  4071 = 'RESET REMAINING\nDOSING VOLUME (ml)' | German: 'RESET RESTDOSIERVOLUMEN (ml)' | France: 'RESET VOLUME DE DOSAGE RESTANT (ml)' | English: 'RESET REMAINING\nDOSING VOLUME (ml)'
  7600 = 'RIGHT\nBOTTOM' | German: 'RECHTS UNTEN' | France: 'DROITE EN BAS' | English: 'RIGHT\nBOTTOM'
  3413 = 'RIGHT\nTOP' | German: 'RECHTS OBEN' | France: 'DROITE EN HAUT' | English: 'RIGHT\nTOP'
  6630 = 'RIGHT BOTTOM TEMP (°C) ' | German: 'TEMPERATUR UNTEN RECHTS' | France: 'TEMPÉRATURE EN BAS À DROITE (?C)' | English: 'RIGHT BOTTOM TEMP (°C) '
  7664 = 'RIGHT TOP TEMP (°C) ' | German: 'TEMPERATUR OBEN RECHTS' | France: 'TEMPÉRATURE EN HAUT À DROITE (?C)' | English: 'RIGHT TOP TEMP (°C) '
  3245 = 'ROTARY BARREL' | German: 'TROMMEL' | France: 'BARILLET ROTATIF' | English: 'ROTARY BARREL'
  4283 = 'ROTARY BARREL - ROBOT' | German: 'TROMMEL - ROTATIONSROBOTER' | France: 'BARILLET ROTATIF - ROBOT DE ROTATION' | English: 'ROTARY BARREL - ROBOT'
  7424 = 'ROTARY BARREL - STATION' | German: 'TROMMEL - WANNE' | France: 'BARILLET ROTATIF - CUVE' | English: 'ROTARY BARREL - STATION'
  2002 = 'ROTATING BARREL' | German: 'TROMMEL' | France: 'BARILLET ROTATIF' | English: 'ROTATING BARREL'
  374 = 'ROW LOADING INC AV-3' | English: 'ROW LOADING INC AV-3'
  6590 = 'ROW MAIN INC AV-2' | English: 'ROW MAIN INC AV-2'
  254 = 'RUN' | German: 'RUN' | France: 'MARCHE' | English: 'RUN'
  5034 = 'SATURDAY' | German: 'SAMSTAG' | France: 'SAMEDI' | English: 'SATURDAY'
  53 = 'SAVE' | German: 'SPEICHERN' | France: 'ENREGISTRER' | English: 'SAVE'
  667 = 'Scan Complete' | German: 'Scan abgeschlossen' | France: 'Scan terminé' | English: 'Scan Complete'
  447 = 'Scan Start' | German: 'Start des Scans' | France: 'Démarrage du scan' | English: 'Scan Start'
  4578 = 'SENSOR A MISSHOOK\nALARM DEACTIVATED' | German: 'SENSOR A FEHLHAKEN\nALARM DEAKTIVIERT' | France: 'DÉTECTEUR A MAL ACCROCHÉ\nALARME DÉSACTIVÉE' | English: 'SENSOR A MISSHOOK\nALARM DEACTIVATED'
  3015 = 'SENSOR B MISSHOOK\nALARM DEACTIVATED' | German: 'SENSOR B FEHLHAKEN\nALARM DEAKTIVIERT' | France: 'DÉTECTEUR B MAL ACCROCHÉ\nALARME DÉSACTIVÉE' | English: 'SENSOR B MISSHOOK\nALARM DEACTIVATED'
  4042 = 'SEQUENCE RECIPE CONFIGURATION (SSER)' | German: 'KONFIGURATION DER SEQUENZREZEPTE (SSER)' | France: 'CONFIGURATION DE LA RECETTE DE SÉQUENCE (SSER)' | English: 'SEQUENCE RECIPE CONFIGURATION (SSER)'
  1305 = 'SEQUENCE RECIPE INFO (SSER)' | German: 'SEQUENZ REZEPTINFO (SSER)' | France: 'INFORMATION SUR LA RECETTE DE LA SÉQUENCE (SSER)' | English: 'SEQUENCE RECIPE INFO (SSER)'
  3694 = 'SET TIME' | German: 'SOLLZEIT' | France: 'TEMPS DE CONSIGNE' | English: 'SET TIME'
  1659 = 'SET VALUE' | German: 'WERT EINSTELLEN' | France: 'DEFINITION DES VALEURS' | English: 'SET VALUE'
  197 = 'SETTING' | German: 'EINSTELLUNG' | France: 'PARAMÈTRES' | English: 'SETTING'
  669 = 'SLOWPULL' | German: 'LIFT OUT' | France: 'SORTIE LENTE' | English: 'SLOWPULL'
  2167 = 'SLOWPULL\nDOWN' | German: 'LIFT OUT\nNACH UNTEN' | France: 'SORTIE LENTE\nNEN BAS' | English: 'SLOWPULL\nDOWN'
  3255 = 'SLOWPULL\nUP' | German: 'LIFT OUT\nNACH ' | France: 'SORTIE LENTE\nHAUT' | English: 'SLOWPULL\nUP'
  4405 = 'SLOWPULL DOWN STN 8' | German: 'LANGSAMES ZIEHEN NACH UNTEN WANNE 8' | France: 'RALENTISSEMENT DE LA DESCENTE AU POSTE 8' | English: 'SLOWPULL DOWN STN 8'
  3314 = 'SLOWPULL JOG VELO (mm/s)' | English: 'SLOWPULL JOG VELO (mm/s)'
  4447 = 'SLOWPULL POSITION' | English: 'SLOWPULL POSITION'
  2433 = 'SLOWPULL VELOCITY (mm/s)' | English: 'SLOWPULL VELOCITY (mm/s)'
  4890 = 'SPEED PATTERN NO' | German: 'GESCHWINDIGKEIT MUSTERNUMMER' | France: 'VITESSE ENTRE POSITION' | English: 'SPEED PATTERN NO'
  4281 = 'SPEED PROFILE NO.' | German: 'GESCHWINDIGKEIT PROFILNUMMER' | France: 'NUMERO DU TYPE DE VITESSE' | English: 'SPEED PROFILE NO.'
  4424 = 'SSER' | German: 'SSER' | France: 'SSER' | English: 'SSER'
  3904 = 'SSER NAME' | German: 'SSER NAME' | France: 'SSER NAME' | English: 'SSER NAME'
  4062 = 'SSER NO.' | German: 'SSER NO.' | France: 'SSER NO.' | English: 'SSER NO.'
  646 = 'SSUR' | German: 'SSUR' | France: 'SSUR' | English: 'SSUR'
  1459 = 'SSUR NAME' | German: 'SSUR NAME' | France: 'SSUR NAME' | English: 'SSUR NAME'
  1820 = 'SSUR NO.' | German: 'SSUR NO.' | France: 'SSUR NO.' | English: 'SSUR NO.'
  224 = 'START' | German: 'START' | France: 'DEMARRER' | English: 'START'
  183 = 'STATION' | German: 'WANNE' | France: 'CUVE' | English: 'STATION'
  370 = 'STATION 01' | German: 'WANNE 01' | France: 'CUVE 01' | English: 'STATION 01'
  742 = 'STATION 02' | German: 'WANNE 02' | France: 'CUVE 02' | English: 'STATION 02'
  859 = 'STATION 03' | German: 'WANNE 03' | France: 'CUVE 03' | English: 'STATION 03'
  200 = 'STATION 04' | German: 'WANNE 04' | France: 'CUVE 04' | English: 'STATION 04'
  72 = 'STATION 05' | German: 'WANNE 05' | France: 'CUVE 05' | English: 'STATION 05'
  509 = 'STATION 06' | German: 'WANNE 06' | France: 'CUVE 06' | English: 'STATION 06'
  120 = 'STATION 07' | German: 'WANNE 07' | France: 'CUVE 07' | English: 'STATION 07'
  712 = 'STATION 08' | German: 'WANNE 08' | France: 'CUVE 08' | English: 'STATION 08'
  1915 = 'STATION 09' | German: 'WANNE 09' | France: 'CUVE 09' | English: 'STATION 09'
  4945 = 'STATION 5 INCOMING WATER' | German: 'WANNE 05 EINGANG VERSORGUNG FÜR WASSER' | France: 'CUVE 05 ALIMENTATION EN EAU ' | English: 'STATION 5 INCOMING WATER'
  3 = 'STATION INFO' | German: 'INFO WANNE' | France: 'INFORMATIONS SUR LA CUVE' | English: 'STATION INFO'
  4252 = 'STATION ROTATION\nBASKET'
  2249 = 'STATION VIEW' | German: 'STATION ANSICHT' | France: 'VUE DE LA STATION' | English: 'STATION VIEW'
  1600 = 'STEP' | German: 'SCHRITTE' | France: 'ETAPE' | English: 'STEP'
  1308 = 'STEP 01' | German: 'SCHRITTE 01' | France: 'ETAPE 01' | English: 'STEP 01'
  541 = 'STEP 02' | German: 'SCHRITTE 02' | France: 'ETAPE 02' | English: 'STEP 02'
  535 = 'STEP 03' | German: 'SCHRITTE 03' | France: 'ETAPE 03' | English: 'STEP 03'
  398 = 'STEP 04' | German: 'SCHRITTE 04' | France: 'ETAPE 04' | English: 'STEP 04'
  1687 = 'STEP 05' | German: 'SCHRITTE 05' | France: 'ETAPE 05' | English: 'STEP 05'
  1286 = 'STEP 06' | German: 'SCHRITTE 06' | France: 'ETAPE 06' | English: 'STEP 06'
  2151 = 'STEP 07' | German: 'SCHRITTE 07' | France: 'ETAPE 07' | English: 'STEP 07'
  1635 = 'STEP 08' | German: 'SCHRITTE 08' | France: 'ETAPE 08' | English: 'STEP 08'
  2165 = 'STEP 09' | German: 'SCHRITTE 09' | France: 'ETAPE 09' | English: 'STEP 09'
  510 = 'STEP 10' | German: 'SCHRITTE 10' | France: 'ETAPE 10' | English: 'STEP 10'
  2122 = 'STEP 11' | German: 'SCHRITTE 11' | France: 'ETAPE 11' | English: 'STEP 11'
  1601 = 'STEP 12' | German: 'SCHRITTE 12' | France: 'ETAPE 12' | English: 'STEP 12'
  1643 = 'STEP 13' | German: 'SCHRITTE 13' | France: 'ETAPE 13' | English: 'STEP 13'
  179 = 'STEP 14' | German: 'SCHRITTE 14' | France: 'ETAPE 14' | English: 'STEP 14'
  2188 = 'STEP 15' | German: 'SCHRITTE 15' | France: 'ETAPE 15' | English: 'STEP 15'
  201 = 'STEP 16' | German: 'SCHRITTE 16' | France: 'ETAPE 16' | English: 'STEP 16'
  1624 = 'STEP 17' | German: 'SCHRITTE 17' | France: 'ETAPE 17' | English: 'STEP 17'
  2332 = 'STEP 18' | German: 'SCHRITTE 18' | France: 'ETAPE 18' | English: 'STEP 18'
  960 = 'STEP 19' | German: 'SCHRITTE 19' | France: 'ETAPE 19' | English: 'STEP 19'
  2078 = 'STEP 20' | German: 'SCHRITTE 20' | France: 'ETAPE 20' | English: 'STEP 20'
  294 = 'STN 01' | German: 'WANNE 01' | France: 'CUVE 01' | English: 'STN 01'
  512 = 'STN 01\nDOWN' | German: 'WANNE 01\nNACH UNTEN' | France: 'CUVE 01\nEN BAS' | English: 'STN 01\nDOWN'
  3517 = 'STN 01\nHOOK' | German: 'WANNE 01\nHAKEN' | France: 'CUVE 01\nACCROCHAGE' | English: 'STN 01\nHOOK'
  2972 = 'STN 01\nUNHOOK' | German: 'WANNE 01\nAUSHANGEN' | France: 'CUVE 01\nDECROCHAGE' | English: 'STN 01\nUNHOOK'
  1354 = 'STN 01 BOTTOM\nSUCTION VALVE AV1-3' | German: 'WANNE 01 DRUCKTASTER\nSAUGLUFTVENTIL 1-3' | France: "CUVE 01 BOUTON-POUSSOIR\nSOUPAPE D'AIR\nD'ASPIRATION 1-3" | English: 'STN 01 BOTTOM\nSUCTION VALVE AV1-3'
  3860 = 'STN 01 BOTTOM\nSUCTION VALVE AV2-3' | German: 'WANNE 01 DRUCKTASTER SAUGLUFTVENTIL 2-3' | France: "CUVE 01 BOUTON-POUSSOIR SOUPAPE D'AIR D'ASPIRATION 2-3" | English: 'STN 01 BOTTOM\nSUCTION VALVE AV2-3'
  8043 = 'STN 01 DIW INC\nSUPPLY VALVE AV1-1' | German: 'WANNE 01 DIW INC\nZUFUHRVENTIL AV1-1' | France: "CUVE 01 DIW INC\nSOUPAPE D'ALIMENTATION\nAV1-1" | English: 'STN 01 DIW INC\nSUPPLY VALVE AV1-1'
  2314 = 'STN 01 DIW INC\nSUPPLY VALVE AV2-1' | German: 'WANNE 01 DIW INC ZUFUHRVENTIL AV2-1' | France: "CUVE 01 DIW INC SOUPAPE D'ALIMENTATION AV2-1" | English: 'STN 01 DIW INC\nSUPPLY VALVE AV2-1'
  474 = 'STN 01 DRAIN' | German: 'WANNE 01 ENTLEERUNG' | France: 'CUVE 01 VIDANGE' | English: 'STN 01 DRAIN'
  1834 = 'STN 01 DRAIN\nVALVE AV1-4' | German: 'WANNE 01 ENTLEERUNG\nSAUGLUFTVENTIL 1-4' | France: "CUVE 01 VIDANGE VANNE\nD'AIR D'ASPIRATION\n1-4" | English: 'STN 01 DRAIN\nVALVE AV1-4'
  1064 = 'STN 01 DRAIN \nVALVE AV1-4' | German: 'WANNE 01 ENTLEERUNG SAUGLUFTVENTIL 1-4' | France: "CUVE 01 VIDANGE VANNE D'AIR D'ASPIRATION 1-4" | English: 'STN 01 DRAIN \nVALVE AV1-4'
  3372 = 'STN 01 DRAIN \nVALVE AV2-4' | German: 'WANNE 01 ENTLEERUNG SAUGLUFTVENTIL 2-4' | France: "CUVE 01 VIDANGE VANNE D'AIR D'ASPIRATION 2-4" | English: 'STN 01 DRAIN \nVALVE AV2-4'
  2307 = 'STN 01 DRAIN  VALVE AV1-4' | German: 'WANNE 01 ENTLEERUNG SAUGLUFTVENTIL 1-4' | France: "CUVE 01 VIDANGE VANNE D'AIR D'ASPIRATION 1-4" | English: 'STN 01 DRAIN  VALVE AV1-4'
  6607 = 'STN 01 DRAIN VALVE AV1-3' | German: 'WANNE 01 ENTLEERUNG\nSAUGLUFTVENTIL 1-3' | France: "CUVE 01 VIDANGE VANNE\nD'AIR D'ASPIRATION 1-3" | English: 'STN 01 DRAIN VALVE AV1-3'
  4935 = 'STN 01 DRAIN VALVE AV1-4' | German: 'WANNE 01 ENTLEERUNG\nSAUGLUFTVENTIL 1-4' | France: "CUVE 01 VIDANGE VANNE\nD'AIR D'ASPIRATION 1-4" | English: 'STN 01 DRAIN VALVE AV1-4'
  4000 = 'STN 01 OVERFLOW\nSUCTION VALVE AV1-2' | German: 'WANNE 01 ÜBERFLUß\nAASAUGUNG VENTIL AV1-2' | France: 'CUVE 01 TROP-PLEIN\nASPIRATION VANNE AV1-2' | English: 'STN 01 OVERFLOW\nSUCTION VALVE AV1-2'
  4585 = 'STN 01 OVERFLOW\nSUCTION VALVE AV2-2' | German: 'WANNE 01 ÜBERFLUß AASAUGUNG VENTIL AV2-3' | France: 'CUVE 01 TROP-PLEIN ASPIRATION VANNE AV2-3' | English: 'STN 01 OVERFLOW\nSUCTION VALVE AV2-2'
  1115 = 'STN 01 PROCESS TANK MIN LEVEL' | German: 'Wanne 01 Niveausensor Prozess - Niveau Minimum' | France: 'CUVE 1 NIVEAU BAS' | English: 'STN 01 PROCESS TANK MIN LEVEL'
  1803 = 'STN 01 READY TEMPERATURE' | German: 'Wanne 01 Bereitschaftstemperatur' | France: 'Cuve 01 Température De Fonctionnement' | English: 'STN 01 READY TEMPERATURE'
  1651 = 'STN 02' | German: 'WANNE 02' | France: 'CUVE 02' | English: 'STN 02'
  2317 = 'STN 02\nDOWN' | German: 'WANNE 02\nNACH UNTEN' | France: 'CUVE 02\nEN BAS' | English: 'STN 02\nDOWN'
  2785 = 'STN 02\nHOOK' | German: 'WANNE 02\nHAKEN' | France: 'CUVE 02\nACCROCHAGE' | English: 'STN 02\nHOOK'
  3442 = 'STN 02\nUNHOOK' | German: 'WANNE 02\nAUSHANGEN' | France: 'CUVE 02\nDECROCHAGE' | English: 'STN 02\nUNHOOK'
  6777 = 'STN 02 BOTTOM\nSUCTION VALVE AV2-3' | German: 'WANNE 02 DRUCKTASTER\nSAUGLUFTVENTIL 2-3' | France: "CUVE 02 BOUTON-POUSSOIR\nSOUPAPE D'AIR\nD'ASPIRATION 2-3" | English: 'STN 02 BOTTOM\nSUCTION VALVE AV2-3'
  3146 = 'STN 02 BOTTOM\nSUCTION VALVE AV2-4' | German: 'WANNE 02 DRUCKTASTER\nSAUGLUFTVENTIL 2-4' | France: "CUVE 02 BOUTON-POUSSOIR\nSOUPAPE D'AIR D'ASPIRATION 2-4" | English: 'STN 02 BOTTOM\nSUCTION VALVE AV2-4'
  731 = 'STN 02 DIW INC\nSUPPLY VALVE AV2-1' | German: 'WANNE 02 DIW INC\nZUFUHRVENTIL AV2-1' | France: "CUVE 02 DIW INC\nSOUPAPE D'ALIMENTATION\nAV2-1" | English: 'STN 02 DIW INC\nSUPPLY VALVE AV2-1'
  4357 = 'STN 02 DRAIN\nVALVE AV2-4' | German: 'WANNE 02 ENTLEERUNG\nSAUGLUFTVENTIL 2-4' | France: "CUVE 02 VIDANGE VANNE\nD'AIR D'ASPIRATION 2-4" | English: 'STN 02 DRAIN\nVALVE AV2-4'
  341 = 'STN 02 DRAIN \nVALVE AV2-4' | German: 'WANNE 02 ENTLEERUNG\nSAUGLUFTVENTIL 2-4' | France: "CUVE 02 VIDANGE VANNE\nD'AIR D'ASPIRATION 2-4" | English: 'STN 02 DRAIN \nVALVE AV2-4'
  194 = 'STN 02 DRAIN VALVE AV1-4' | German: 'WANNE 02 ENTLEERUNG\nSAUGLUFTVENTIL 1-4' | France: "CUVE 02 VIDANGE VANNE\nD'AIR D'ASPIRATION 1-4" | English: 'STN 02 DRAIN VALVE AV1-4'
  3264 = 'STN 02 INC\nSUPPLY VALVE AV2-1' | German: 'WANNE 02 DIW INC\nZUFUHRVENTIL AV2-1' | France: "CUVE 02 DIW INC\nSOUPAPE D'ALIMENTATION\nAV2-1" | English: 'STN 02 INC\nSUPPLY VALVE AV2-1'
  6735 = 'STN 02 OVERFLOW\nSUCTION VALVE AV2-2' | German: 'WANNE 02 ÜBERFLUß AASAUGUNG VENTIL AV2-2' | France: 'CUVE 02 TROP-PLEIN\nASPIRATION VANNE AV2-2' | English: 'STN 02 OVERFLOW\nSUCTION VALVE AV2-2'
  3083 = 'STN 02 OVERFLOW \nSUCTION VALVE AV2-2\n' | German: 'WANNE 02 ÜBERFLUß\nAASAUGUNG VENTIL AV2-2' | France: 'CUVE 02 TROP-PLEIN\nASPIRATION VANNE AV2-2' | English: 'STN 02 OVERFLOW \nSUCTION VALVE AV2-2\n'
  1861 = 'STN 02 PROCESS TANK MIN LEVEL' | German: 'Wanne 02 Niveausensor Prozess - Niveau Minimum' | France: 'CUVE 2 NIVEAU BAS' | English: 'STN 02 PROCESS TANK MIN LEVEL'
  2860 = 'STN 02 READY TEMPERATURE' | German: 'Wanne 02 Bereitschaftstemperatur' | France: 'Cuve 02 Température De Fonctionnement' | English: 'STN 02 READY TEMPERATURE'
  1227 = 'STN 02 ROW INC\nSUPPLY VALVE AV2-1' | English: 'STN 02 ROW INC\nSUPPLY VALVE AV2-1'
  813 = 'STN 03' | German: 'WANNE 03' | France: 'CUVE 03' | English: 'STN 03'
  1393 = 'STN 03\nDOWN' | German: 'WANNE 03\nNACH UNTEN' | France: 'CUVE 03\nEN BAS' | English: 'STN 03\nDOWN'
  3367 = 'STN 03\nHOOK' | German: 'WANNE 03\nHAKEN' | France: 'CUVE 03\nACCROCHAGE' | English: 'STN 03\nHOOK'
  4177 = 'STN 03\nUNHOOK' | German: 'WANNE 03\nAUSHANGEN' | France: 'CUVE 03\nDECROCHAGE' | English: 'STN 03\nUNHOOK'
  4961 = 'STN 03 BOTTOM\nSUCTION VALVE AV3-3' | German: 'WANNE 03 DRUCKTASTER\nSAUGLUFTVENTIL 3-3' | France: "CUVE 03 BOUTON-POUSSOIR\nSOUPAPE D'AIR\nD'ASPIRATION 3-3" | English: 'STN 03 BOTTOM\nSUCTION VALVE AV3-3'
  723 = 'STN 03 BOTTOM\nSUCTION VALVE AV4-3' | German: 'WANNE 03 DRUCKTASTER\nSAUGLUFTVENTIL 3-4' | France: "CUVE 03 BOUTON-POUSSOIR\nSOUPAPE D'AIR\nD'ASPIRATION 3-4" | English: 'STN 03 BOTTOM\nSUCTION VALVE AV4-3'
  8217 = 'STN 03 DIW INC\nSUPPLY VALVE AV3-1' | German: 'WANNE 03 DIW INC\nZUFUHRVENTIL AV3-1' | France: "CUVE 03 DIW INC\nSOUPAPE D'ALIMENTATION\nAV3-1" | English: 'STN 03 DIW INC\nSUPPLY VALVE AV3-1'
  4960 = 'STN 03 DRAIN\nVALVE AV3-4' | German: 'WANNE 03 ENTLEERUNG\nSAUGLUFTVENTIL 3-4' | France: "CUVE 03 VIDANGE VANNE\nD'AIR D'ASPIRATION 3-4" | English: 'STN 03 DRAIN\nVALVE AV3-4'
  6707 = 'STN 03 DRAIN\nVALVE AV4-4' | German: 'WANNE 03 ENTLEERUNG SAUGLUFTVENTIL 3-4' | France: "CUVE 03 VIDANGE VANNE\nD'AIR D'ASPIRATION 3-4" | English: 'STN 03 DRAIN\nVALVE AV4-4'
  1570 = 'STN 03 DRAIN \nVALVE AV3-4' | German: 'WANNE 03 ENTLEERUNG SAUGLUFTVENTIL 3-4' | France: "CUVE 03 VIDANGE VANNE\nD'AIR D'ASPIRATION 3-4" | English: 'STN 03 DRAIN \nVALVE AV3-4'
  979 = 'STN 03 INC\nSUPPLY VALVE AV3-1' | German: 'WANNE 03 DIW INC\nZUFUHRVENTIL AV3-1' | France: "CUVE 03 DIW INC\nSOUPAPE D'ALIMENTATION AV3-1" | English: 'STN 03 INC\nSUPPLY VALVE AV3-1'
  7506 = 'STN 03 INC\nSUPPLY VALVE AV4-1' | German: 'WANNE 03 DIW INC\nZUFUHRVENTIL AV4-1' | France: "CUVE 03 DIW INC\nSOUPAPE D'ALIMENTATION AV4-1" | English: 'STN 03 INC\nSUPPLY VALVE AV4-1'
  8087 = 'STN 03 OVERFLOW\nSUCTION VALVE AV3-2' | German: 'WANNE 03 ÜBERFLUß\nAASAUGUNG VENTIL AV3-2' | France: 'CUVE 03 TROP-PLEIN\nASPIRATION VANNE AV3-2' | English: 'STN 03 OVERFLOW\nSUCTION VALVE AV3-2'
  7190 = 'STN 03 OVERFLOW \nSUCTION VALVE AV3-2\n' | German: 'WANNE 03 ÜBERFLUß\nAASAUGUNG VENTIL AV2-2' | France: 'CUVE 03 TROP-PLEIN\nASPIRATION VANNE AV3-2' | English: 'STN 03 OVERFLOW \nSUCTION VALVE AV3-2\n'
  5431 = 'STN 03 OVERFLOW \nSUCTION VALVE AV4-2\n' | German: 'WANNE 02 ÜBERFLUß\nAASAUGUNG VENTIL AV2-3' | France: 'CUVE 03 TROP-PLEIN\nASPIRATION VANNE AV2-3' | English: 'STN 03 OVERFLOW \nSUCTION VALVE AV4-2\n'
  949 = 'STN 03 PROCESS TANK MIN LEVEL' | German: 'Wanne 03 Niveausensor Prozess - Niveau Minimum' | France: 'CUVE 3 NIVEAU BAS' | English: 'STN 03 PROCESS TANK MIN LEVEL'
  337 = 'STN 03 READY TEMPERATURE' | German: 'Wanne 03 Bereitschaftstemperatur' | France: 'Cuve 03 Température De Fonctionnement' | English: 'STN 03 READY TEMPERATURE'
  2144 = 'STN 04' | German: 'WANNE 04' | France: 'CUVE 04' | English: 'STN 04'
  4423 = 'STN 04\nDOWN' | German: 'WANNE 04\nNACH UNTEN' | France: 'CUVE 04\nEN BAS' | English: 'STN 04\nDOWN'
  1019 = 'STN 04\nHOOK' | German: 'WANNE 04\nHAKEN' | France: 'CUVE 04\nACCROCHAGE' | English: 'STN 04\nHOOK'
  2377 = 'STN 04\nUNHOOK' | German: 'WANNE 04\nAUSHANGEN' | France: 'CUVE 04\nDECROCHAGE' | English: 'STN 04\nUNHOOK'
  4758 = 'STN 04 BOTTOM\nSUCTION VALVE AV4-3' | German: 'WANNE 04 DRUCKTASTER\nSAUGLUFTVENTIL 4-3' | France: "CUVE 04 BOUTON-POUSSOIR\nSOUPAPE D'AIR\nD'ASPIRATION 4-3" | English: 'STN 04 BOTTOM\nSUCTION VALVE AV4-3'
  6731 = 'STN 04 DIW INC\nSUPPLY VALVE AV4-1' | German: 'WANNE 04 DIW INC\nZUFUHRVENTIL AV4-1' | France: "CUVE 04 DIW INC\nSOUPAPE D'ALIMENTATION\nAV4-1" | English: 'STN 04 DIW INC\nSUPPLY VALVE AV4-1'
  6404 = 'STN 04 DRAIN\nVALVE AV4-4' | German: 'WANNE 04 ENTLEERUNG\nSAUGLUFTVENTIL 4-4' | France: "CUVE 04 VIDANGE VANNE\nD'AIR D'ASPIRATION 4-4" | English: 'STN 04 DRAIN\nVALVE AV4-4'
  6821 = 'STN 04 DRAIN\nVALVE AV5-4' | German: 'WANNE 04 ENTLEERUNG\nSAUGLUFTVENTIL 5-4' | France: "CUVE 04 VIDANGE VANNE D'AIR\nD'ASPIRATION 4-4" | English: 'STN 04 DRAIN\nVALVE AV5-4'
  2015 = 'STN 04 DRAIN \nVALVE AV4-4' | German: 'WANNE 04 ENTLEERUNG\nSAUGLUFTVENTIL 4-4' | France: "CUVE 04 VIDANGE VANNE D'AIR\nD'ASPIRATION 4-4" | English: 'STN 04 DRAIN \nVALVE AV4-4'
  1560 = 'STN 04 INC\nSUPPLY VALVE AV4-1' | German: 'WANNE 04 DIW INC\nZUFUHRVENTIL AV4-1' | France: "CUVE 04 DIW INC\nSOUPAPE D'ALIMENTATION AV4-1" | English: 'STN 04 INC\nSUPPLY VALVE AV4-1'
  2047 = 'STN 04 OVERFLOW\nSUCTION VALVE AV4-2' | German: 'WANNE 04 ÜBERFLUß\nAASAUGUNG VENTIL AV4-2' | France: 'CUVE 04 TROP-PLEIN\nASPIRATION VANNE AV4-2' | English: 'STN 04 OVERFLOW\nSUCTION VALVE AV4-2'
  5099 = 'STN 04 OVERFLOW \nSUCTION VALVE AV4-2\n' | German: 'WANNE 04 ÜBERFLUß\nAASAUGUNG VENTIL AV4-2' | France: 'CUVE 04 TROP-PLEIN\nASPIRATION VANNE AV4-2' | English: 'STN 04 OVERFLOW \nSUCTION VALVE AV4-2\n'
  1508 = 'STN 04 PROCESS TANK MIN LEVEL' | German: 'Wanne 04 Niveausensor Prozess - Niveau Minimum' | France: 'CUVE 4 NIVEAU BAS' | English: 'STN 04 PROCESS TANK MIN LEVEL'
  1561 = 'STN 04 READY TEMPERATURE' | German: 'Wanne 04 Bereitschaftstemperatur' | France: 'Cuve 04 Température De Fonctionnement' | English: 'STN 04 READY TEMPERATURE'
  6412 = 'STN 04 ROW INC\nSUPPLY VALVE AV4-1' | English: 'STN 04 ROW INC\nSUPPLY VALVE AV4-1'
  1110 = 'STN 05' | German: 'WANNE 05' | France: 'CUVE 05' | English: 'STN 05'
  1404 = 'STN 05\nDOWN' | German: 'WANNE 05\nNACH UNTEN' | France: 'CUVE 05\nEN BAS' | English: 'STN 05\nDOWN'
  450 = 'STN 05\nHOOK' | German: 'WANNE 05\nHAKEN' | France: 'CUVE 05\nACCROCHAGE' | English: 'STN 05\nHOOK'
  275 = 'STN 05\nUNHOOK' | German: 'WANNE 05\nAUSHANGEN' | France: 'CUVE 05\nDECROCHAGE' | English: 'STN 05\nUNHOOK'
  371 = 'STN 05 BOTTOM\nSUCTION VALVE AV4-3' | German: 'WANNE 05 DRUCKTASTER\nSAUGLUFTVENTIL 4-3' | France: "CUVE 05 BOUTON-POUSSOIR\nSOUPAPE D'AIR D'ASPIRATION 4-3" | English: 'STN 05 BOTTOM\nSUCTION VALVE AV4-3'
  6465 = 'STN 05 BOTTOM\nSUCTION VALVE AV5-3' | German: 'WANNE 05 DRUCKTASTER\nSAUGLUFTVENTIL 5-3' | France: "CUVE 05 BOUTON-POUSSOIR\nSOUPAPE D'AIR D'ASPIRATION 5-3" | English: 'STN 05 BOTTOM\nSUCTION VALVE AV5-3'
  5882 = 'STN 05 DIW INC\nSUPPLY VALVE AV5-1' | German: 'WANNE 05 DIW INC\nZUFUHRVENTIL AV5-1' | France: "CUVE 05 DIW INC\nSOUPAPE D'ALIMENTATION\nAV5-1" | English: 'STN 05 DIW INC\nSUPPLY VALVE AV5-1'
  4563 = 'STN 05 DRAIN \nVALVE AV5-4' | German: 'WANNE 05 ENTLEERUNG\nSAUGLUFTVENTIL 5-4' | France: "CUVE 05 VIDANGE VANNE\nD'AIR D'ASPIRATION 5-4" | English: 'STN 05 DRAIN \nVALVE AV5-4'
  6510 = 'STN 05 INC\nSUPPLY VALVE AV4-1' | German: 'WANNE 05 DIW INC\nZUFUHRVENTIL AV4-1' | France: "CUVE 04 DIW INC SOUPAPE\nD'ALIMENTATION AV4-1" | English: 'STN 05 INC\nSUPPLY VALVE AV4-1'
  1680 = 'STN 05 INC\nSUPPLY VALVE AV5-1' | German: 'WANNE 05 DIW INC\nZUFUHRVENTIL AV5-1' | France: "CUVE 05 DIW INC SOUPAPE\nD'ALIMENTATION AV5-1" | English: 'STN 05 INC\nSUPPLY VALVE AV5-1'
  7483 = 'STN 05 INCOMING\nDIW SUPPLY AV5-1' | German: 'WANNE 05 DIW INC\nZUFUHRVENTIL AV5-1' | France: "CUVE 05 DIW INC SOUPAPE\nD'ALIMENTATION AV5-1" | English: 'STN 05 INCOMING\nDIW SUPPLY AV5-1'
  8763 = 'STN 05 INCOMING CW \nSUPPLY AV5-2'
  387 = 'STN 05 INCOMING CW \nSUPPLY AV5-2\n' | German: 'WANNE 05 CW INC\nZUFUHRVENTIL AV5-2' | France: "CUVE 05 CW INC SOUPAPE\nD'ALIMENTATION AV5-2" | English: 'STN 05 INCOMING CW \nSUPPLY AV5-2\n'
  2356 = 'STN 05 OVERFLOW\nSUCTION VALVE AV5-2' | German: 'WANNE 05 ÜBERFLUß\nAASAUGUNG VENTIL AV5-2' | France: 'CUVE 05 TROP-PLEIN\nASPIRATION VANNE AV5-2' | English: 'STN 05 OVERFLOW\nSUCTION VALVE AV5-2'
  2606 = 'STN 05 OVERFLOW \nSUCTION VALVE AV4-2\n' | German: 'WANNE 05 ÜBERFLUß\nAASAUGUNG VENTIL AV4-2' | France: 'CUVE 05 TROP-PLEIN\nASPIRATION VANNE AV4-2' | English: 'STN 05 OVERFLOW \nSUCTION VALVE AV4-2\n'
  5340 = 'STN 05 OVERFLOW \nSUCTION VALVE AV5-2\n' | German: 'WANNE 05 ÜBERFLUß\nAASAUGUNG VENTIL AV5-2' | France: 'CUVE 05 TROP-PLEIN\nASPIRATION VANNE AV5-2' | English: 'STN 05 OVERFLOW \nSUCTION VALVE AV5-2\n'
  986 = 'STN 05 PROCESS TANK MIN LEVEL' | German: 'Wanne 05 Niveausensor Prozess - Niveau Minimum' | France: 'CUVE 5 NIVEAU BAS' | English: 'STN 05 PROCESS TANK MIN LEVEL'
  3351 = 'STN 05 READY TEMPERATURE' | German: 'Wanne 05 Bereitschaftstemperatur' | France: 'Cuve 05 Température De Fonctionnement' | English: 'STN 05 READY TEMPERATURE'
  436 = 'STN 06' | German: 'WANNE 06' | France: 'CUVE 06' | English: 'STN 06'
  4491 = 'STN 06\nDOOR CLAMP' | German: 'WANNE 06\nSCHIEBETÜR GESCHLOSSEN' | France: 'CUVE 06\nPORTES COULISSANTES - FERMÉ' | English: 'STN 06\nDOOR CLAMP'
  5348 = 'STN 06\nDOOR CLOSE' | German: 'WANNE 06\nSCHIEBETÜR SCHLIESSEN' | France: 'CUVE 06\nPORTE FERMEE' | English: 'STN 06\nDOOR CLOSE'
  2327 = 'STN 06\nDOOR CLOSED' | German: 'WANNE 06\nSCHIEBETÜR SCHLIESSEN' | France: 'CUVE 06\nPORTE FERMEE' | English: 'STN 06\nDOOR CLOSED'
  6314 = 'STN 06\nDOOR OPEN' | German: 'WANNE 06 SCHIEBEDECKEL ÖFFNEN' | France: 'COUVERCLE COULISSANT CUVE 6 OUV' | English: 'STN 06\nDOOR OPEN'
  4822 = 'STN 06\nDOOR UNCLAMP' | German: 'WANNE 06\nSCHIEBETÜR GEÖFFNET' | France: 'CUVE 06\nPORTES COULISSANTES - OUVERT' | English: 'STN 06\nDOOR UNCLAMP'
  2916 = 'STN 06\nDOWN' | German: 'WANNE 06\nNACH UNTEN' | France: 'CUVE 06\nEN BAS' | English: 'STN 06\nDOWN'
  3548 = 'STN 06\nHOOK' | German: 'WANNE 06\nHAKEN' | France: 'CUVE 06\nACCROCHAGE' | English: 'STN 06\nHOOK'
  1817 = 'STN 06\nUNHOOK' | German: 'WANNE 06\nAUSHANGEN' | France: 'CUVE 06\nDECROCHAGE' | English: 'STN 06\nUNHOOK'
  1963 = 'STN 06 BLOWER \nPROTECTION AV6-1' | German: 'WANNE 06 GEBLÄSESCHUTZ\nSAUGLUFTVENTIL 6-1' | France: "CUVE 06 PROTECTION\nDU VENTILATEUR SOUPAPE\nD'AIR D'ASPIRATION 6-1" | English: 'STN 06 BLOWER \nPROTECTION AV6-1'
  7026 = 'STN 06 BLOWER \nPROTECTION AV6-1\n' | German: 'WANNE 06 GEBLÄSESCHUTZ\nSAUGLUFTVENTIL 6-1' | France: "CUVE 06 PROTECTION\nDU VENTILATEUR SOUPAPE\nD'AIR D'ASPIRATION 6-1" | English: 'STN 06 BLOWER \nPROTECTION AV6-1\n'
  6675 = 'STN 06 BLOWER \nPROTECTION AV6-2' | German: 'WANNE 06 GEBLÄSESCHUTZ\nSAUGLUFTVENTIL 6-2' | France: "CUVE 06 PROTECTION\nDU VENTILATEUR SOUPAPE\nD'AIR D'ASPIRATION 6-2" | English: 'STN 06 BLOWER \nPROTECTION AV6-2'
  7223 = 'STN 06 BLOWER \nPROTECTION AV6-2\n' | German: 'WANNE 06 GEBLÄSESCHUTZ\nSAUGLUFTVENTIL 6-2' | France: "CUVE 06 PROTECTION\nDU VENTILATEUR SOUPAPE\nD'AIR D'ASPIRATION 6-2" | English: 'STN 06 BLOWER \nPROTECTION AV6-2\n'
  4781 = 'STN 06 BLOWER \nPROTECTION VALVE AV6-2\n' | German: 'WANNE 06 GEBLÄSESCHUTZ\nSAUGLUFTVENTIL 6-2' | France: "CUVE 06 PROTECTION\nDU VENTILATEUR SOUPAPE\nD'AIR D'ASPIRATION 6-2" | English: 'STN 06 BLOWER \nPROTECTION VALVE AV6-2\n'
  6784 = 'STN 06 OVERFLOW \nSUCTION VALVE AV5-2\n' | German: 'WANNE 06 ÜBERFLUß AASAUGUNG VENTIL AV5-2' | France: 'CUVE 06 TROP-PLEIN ASPIRATION VANNE AV5-2' | English: 'STN 06 OVERFLOW \nSUCTION VALVE AV5-2\n'
  2381 = 'STN 06 PROCESS TANK MIN LEVEL' | German: 'Wanne 06 Niveausensor Prozess - Niveau Minimum' | France: 'CUVE 6 NIVEAU BAS' | English: 'STN 06 PROCESS TANK MIN LEVEL'
  547 = 'STN 06 READY TEMPERATURE' | German: 'Wanne 06 Bereitschaftstemperatur' | France: 'Cuve 06 Température De Fonctionnement' | English: 'STN 06 READY TEMPERATURE'
  6228 = 'STN 06 ROW INC\nSUPPLY VALVE AV6-1' | English: 'STN 06 ROW INC\nSUPPLY VALVE AV6-1'
  1244 = 'STN 06 ROW INC\nSUPPLY VALVE AV6-2' | English: 'STN 06 ROW INC\nSUPPLY VALVE AV6-2'
  503 = 'STN 06 VACUUM\nRELEASE VALVE AV6-4' | German: 'WANNE 06 VAKUUMENTLÜFTUNG\nSAUGLUFTVENTIL 6-4' | France: 'CUVE 06 VACUUM VENTILATION\nSUCTION AIR VALVE 6-4' | English: 'STN 06 VACUUM\nRELEASE VALVE AV6-4'
  6852 = 'STN 06 VACUUM\nSUCTION VALVE AV5-3' | German: 'WANNE 06 VAKUUMABSAUGUNG\nSAUGLUFTVENTIL 5-3' | France: 'CUVE 06 VACUUM VENTILATION\nSUCTION AIR VALVE 5-4' | English: 'STN 06 VACUUM\nSUCTION VALVE AV5-3'
  8004 = 'STN 06 VACUUM\nSUCTION VALVE AV6-3' | German: 'WANNE 06 VAKUUMABSAUGUNG\nSAUGLUFTVENTIL 6-3' | France: "CUVE 06 ASPIRATION\nSOUS VIDE SOUPAPE\nD'AIR D'ASPIRATION 6-3" | English: 'STN 06 VACUUM\nSUCTION VALVE AV6-3'
  1045 = 'STN 07' | German: 'WANNE 07' | France: 'CUVE 07' | English: 'STN 07'
  3629 = 'STN 07\nDOWN' | German: 'WANNE 07\nNACH UNTEN' | France: 'CUVE 07\nEN BAS' | English: 'STN 07\nDOWN'
  3382 = 'STN 07\nHOOK' | German: 'WANNE 07\nHAKEN' | France: 'CUVE 07\nACCROCHAGE' | English: 'STN 07\nHOOK'
  4206 = 'STN 07\nUNHOOK' | German: 'WANNE 07\nAUSHANGEN' | France: 'CUVE 07\nDECROCHAGE' | English: 'STN 07\nUNHOOK'
  2658 = 'STN 07 PROCESS TANK MIN LEVEL' | German: 'WANNE 07 NIVEAUSENSOR PROZESS - NIVEAU MINIMUM' | France: 'CUVE 7 NIVEAU BAS' | English: 'STN 07 PROCESS TANK MIN LEVEL'
  2156 = 'STN 07 READY TEMPERATURE' | German: 'WANNE 07 BEREITSCHAFTSTEMPERATUR' | France: 'CUVE 07 TEMPÉRATURE DE FONCTIONNEMENT' | English: 'STN 07 READY TEMPERATURE'
  607 = 'STN 08' | German: 'WANNE 08' | France: 'CUVE 08' | English: 'STN 08'
  491 = 'STN 08\nDOWN' | German: 'WANNE 08\nNACH UNTEN' | France: 'CUVE 08\nEN BAS' | English: 'STN 08\nDOWN'
  1410 = 'STN 08\nHOOK' | German: 'WANNE 08\nHAKEN' | France: 'CUVE 08\nACCROCHAGE' | English: 'STN 08\nHOOK'
  1838 = 'STN 08\nMID DOWN' | English: 'STN 08\nMID DOWN'
  3387 = 'STN 08\nUNHOOK' | German: 'WANNE 08\nAUSHANGEN' | France: 'CUVE 08\nDECROCHAGE' | English: 'STN 08\nUNHOOK'
  2204 = 'STN 08 PROCESS TANK MIN LEVEL' | German: 'WANNE 08 NIVEAUSENSOR PROZESS - NIVEAU MINIMUM' | France: 'CUVE 8 NIVEAU BAS' | English: 'STN 08 PROCESS TANK MIN LEVEL'
  2501 = 'STN 09' | German: 'WANNE 09' | France: 'CUVE 09' | English: 'STN 09'
  1986 = 'STN 09\nDOWN' | German: 'WANNE 09\nNACH UNTEN' | France: 'CUVE 09\nEN BAS' | English: 'STN 09\nDOWN'
  2340 = 'STN 09\nHOOK' | German: 'WANNE 09\nHAKEN' | France: 'CUVE 09\nACCROCHAGE' | English: 'STN 09\nHOOK'
  520 = 'STN 09\nUNHOOK' | German: 'WANNE 09\nAUSHANGEN' | France: 'CUVE 09\nDECROCHAGE' | English: 'STN 09\nUNHOOK'
  5755 = 'STN 1-4 CHEMICAL RETURN TANK PUMP' | German: 'WANNE 01 - 04 PUMPE FÜR CHEMIKALIENRÜCKLAUFTANK' | France: 'CUVE 01 - 04 POMPE DE RETOUR DE PRODUITS CHIMIQUES ' | English: 'STN 1-4 CHEMICAL RETURN TANK PUMP'
  4920 = 'STN 1-4 EXHAUST BLOWER' | German: 'WANNE 01 - 06 ABLUFTGEBLÄSE' | France: "CUVE 01 - 06 VENTILATEUR D'EXTRACTION" | English: 'STN 1-4 EXHAUST BLOWER'
  3161 = 'STN 1-5 AGITATION MOTOR' | German: 'WANNE 01 - 05 MOTOR WARENBEWEGUNG ' | France: 'CUVE 01 - 05 MOTEUR MOUVEMENT DU PRODUIT' | English: 'STN 1-5 AGITATION MOTOR'
  892 = 'STN 1-6 EXHAUST\nBLOWER' | German: 'WANNE 01 - 06 ABLUFTGEBLÄSE' | France: "CUVE 01 - 06 VENTILATEUR D'EXTRACTION" | English: 'STN 1-6 EXHAUST\nBLOWER'
  7438 = 'STN 1-6 EXHAUST BLOWER' | German: 'WANNE 01 - 06 ABLUFTGEBLÄSE' | France: "CUVE 01 - 06 VENTILATEUR D'EXTRACTION" | English: 'STN 1-6 EXHAUST BLOWER'
  7816 = 'STN 1-7 AGITATION MOTOR' | German: 'WANNE 01 - 05 MOTOR WARENBEWEGUNG ' | France: 'CUVE 01 - 05 MOTEUR MOUVEMENT DU PRODUIT' | English: 'STN 1-7 AGITATION MOTOR'
  6439 = 'STN 5-6 FFU ' | German: 'WANNE 05 - 06 FILTER EINHEIT ' | France: 'CUVE 05 - 06 UNITÉ DE FILTRE ' | English: 'STN 5-6 FFU '
  7765 = 'STN 5-6 FFU UNIT' | German: 'WANNE 05 - 06 FILTER EINHEIT ' | France: 'CUVE 05 - 06 UNITÉ DE FILTRE ' | English: 'STN 5-6 FFU UNIT'
  3373 = 'STN 8 SLOW PULL' | English: 'STN 8 SLOW PULL'
  633 = 'STOP' | German: 'HALT' | France: 'ARRET' | English: 'STOP'
  664 = 'SUB PROCESS RECIPE CONFIGURATION (SSUR)' | German: 'KONFIGURATION DER SUBPROZESSREZEPTE' | France: 'CONFIGURATION DE LA RECETTE DE SOUS-PROCESSUS (SSUR)' | English: 'SUB PROCESS RECIPE CONFIGURATION (SSUR)'
  2224 = 'SUB PROCESS RECIPE INFO (SSUR)' | German: 'INFO DER SUBPROZESSREZEPTE' | France: 'INFO SUR LES RECETTES DE SOUS-PROCESSUS (SSUR)' | English: 'SUB PROCESS RECIPE INFO (SSUR)'
  1574 = 'SUNDAY' | German: 'SONNTAG' | France: 'DIMANCHE' | English: 'SUNDAY'
  2871 = 'SV' | German: 'SV' | France: 'SV' | English: 'SV'
  1513 = 'TAKT TIMER (sec)' | German: 'TAKT TIMER (Sek.)' | France: 'TAKT TIMER (sec)' | English: 'TAKT TIMER (sec)'
  660 = 'TANK TEMPERATURE (°C)' | German: 'WANNE TEMPERATUR(°C)' | France: 'CUVE TEMPERATURE' | English: 'TANK TEMPERATURE (°C)'
  10007 = 'TEMP NOT READY ALARM' | German: 'ALARM TEMPERATUR NOK' | France: 'ALARME TEMPÉRATURE NON PRÊTE' | English: 'TEMP NOT READY ALARM'
  7215 = 'TEMP PV (°C)  ' | German: 'TEMPERATUR VALEUR REELLE' | France: 'TEMPERATURE ACTUEL' | English: 'TEMP PV (°C)  '
  567 = 'TEMPERATURE' | German: 'TEMPERATUR' | France: 'TEMPERATURE' | English: 'TEMPERATURE'
  4669 = 'THURSDAY' | German: 'DONNERSTAG' | France: 'JEUDI' | English: 'THURSDAY'
  8390 = 'TIME OPTIMIZE/TRACKER' | German: 'ZEITOPTIMIERUNG/TRACKER' | France: 'OPTIMISATION DU TEMPS/TRACEUR' | English: 'TIME OPTIMIZE/TRACKER'
  5394 = 'TIMER (sec)' | German: 'ZEITSCHALTUNG (Sek.)' | France: 'MINUTERIE (sec.)' | English: 'TIMER (sec)'
  1727 = 'TO' | German: 'ZU' | France: 'TO' | English: 'TO'
  573 = 'TOP' | German: 'OBEN' | France: 'HAUT' | English: 'TOP'
  3738 = 'TOP POSITION' | German: 'SPITZEN POSITION' | France: 'HAUT CUVE' | English: 'TOP POSITION'
  222 = 'TOTAL' | German: 'SUMMERNZAHLER' | France: 'TOTALE' | English: 'TOTAL'
  5188 = 'TOTALIZER DOSING\nVOLUME' | German: 'ZÄHLWERK\nDOSIERVOLUMEN' | France: 'TOTALISATEUR DU\nVOLUME DE DOSAGE' | English: 'TOTALIZER DOSING\nVOLUME'
  2552 = 'TOTALIZER DOSING\nVOLUME (ml)' | German: 'ZÄHLWERK\nDOSIERVOLUMEN (ml)' | France: 'TOTALISATEUR DU\nVOLUME DE DOSAGE\n(ml)' | English: 'TOTALIZER DOSING\nVOLUME (ml)'
  730 = 'Tracker In progress' | German: 'Tracker In Bearbeitung' | France: 'Tracker en cours' | English: 'Tracker In progress'
  1022 = 'Tracker Info Available' | German: 'Tracker-Informationen verfügbar' | France: 'Informations disponibles sur le traceur' | English: 'Tracker Info Available'
  3941 = 'Tracker Info Not Available' | German: 'Tracker-Informationen nicht verfügbar' | France: 'Informations indisponibles sur le traceur' | English: 'Tracker Info Not Available'
  3628 = 'TUESDAY' | German: 'DIENSTAG' | France: 'MARDI' | English: 'TUESDAY'
  4190 = 'ULD\nDOOR CLOSED' | English: 'ULD\nDOOR CLOSED'
  4290 = 'ULD\nDOOR OPEN' | English: 'ULD\nDOOR OPEN'
  1934 = 'ULD\nDOWN' | English: 'ULD\nDOWN'
  1088 = 'ULD\nHOOK' | English: 'ULD\nHOOK'
  935 = 'ULD\nUNHOOK' | English: 'ULD\nUNHOOK'
  2464 = 'ULD CONVEYOR\nDOOR CLOSED' | English: 'ULD CONVEYOR\nDOOR CLOSED'
  1016 = 'ULD CONVEYOR\nDOOR OPEN' | English: 'ULD CONVEYOR\nDOOR OPEN'
  3020 = 'ULD CONVEYOR MOTOR 1' | English: 'ULD CONVEYOR MOTOR 1'
  5931 = 'ULD CONVEYOR MOTOR 2' | English: 'ULD CONVEYOR MOTOR 2'
  513 = 'ULD CONVEYOR MOTOR 3' | English: 'ULD CONVEYOR MOTOR 3'
  1366 = 'ULD CONVEYOR MOTOR 4' | English: 'ULD CONVEYOR MOTOR 4'
  2917 = 'ULTRASONIC' | German: 'ULTRASCHALL' | France: 'ULTRASONS' | English: 'ULTRASONIC'
  4066 = 'ULTRASONIC ' | German: 'ULTRASCHALL' | France: 'ULTRASONS' | English: 'ULTRASONIC '
  5782 = 'ULTRASONIC BOTTOM' | German: 'ULTRASCHALL UNTEN' | France: 'ULTRASONS DU FOND ' | English: 'ULTRASONIC BOTTOM'
  1471 = 'ULTRASONIC BOTTOM FREQ (kHz)' | German: 'ULTRASCHALL-UNTERFREQUENZ(kHz)' | France: 'FRÉQUENCE ULTRASONS DU FOND ' | English: 'ULTRASONIC BOTTOM FREQ (kHz)'
  2017 = 'ULTRASONIC BOTTOM POWER (%)' | German: 'ULTRASCHALL-UNTERLEISTUNG(%)' | France: 'FOND ULTRASONS PUISSANT' | English: 'ULTRASONIC BOTTOM POWER (%)'
  7723 = 'ULTRASONIC FREQ (kHz)' | German: 'ULTRASCHALL-FREQUENZ(kHz)' | France: 'FRÉQUENCE ULTRASONS' | English: 'ULTRASONIC FREQ (kHz)'
  2282 = 'ULTRASONIC POWER (%)' | German: 'ULTRASCHALL-LEISTUNG(%)' | France: 'PUISSANCE ULTRASONS' | English: 'ULTRASONIC POWER (%)'
  874 = 'ULTRASONIC SIDE' | German: 'ULTRASCHALLSEITE' | France: 'ULTRASONS COTE' | English: 'ULTRASONIC SIDE'
  1578 = 'ULTRASONIC SIDE FREQ (kHz)' | German: 'ULTRASCHALL-SEITENFREQUENZ(kHz)' | France: 'FRÉQUENCE ULTRASONS CÔTÉ ' | English: 'ULTRASONIC SIDE FREQ (kHz)'
  2764 = 'ULTRASONIC SIDE POWER (%)' | German: 'ULTRASCHALLSEITIGE LEISTUNG(%)' | France: 'CÔTÉ ULTRASONS DE PUISSANCE' | English: 'ULTRASONIC SIDE POWER (%)'
  3204 = 'ULTRASONIC SONIC' | German: 'ULTRASCHALL' | France: 'ULTRASONS' | English: 'ULTRASONIC SONIC'
  2639 = 'UNHOOK' | German: 'AUSHANGEN' | France: 'DECROCHAGE' | English: 'UNHOOK'
  24 = 'UNLOADING' | German: 'ENTLADEN' | France: 'DECHARGEMENT' | English: 'UNLOADING'
  2520 = 'UNLOADING BUZZER' | German: 'ENTLADE-SUMMER' | France: 'BUZZER DE DÉCHARGEMENT' | English: 'UNLOADING BUZZER'
  2072 = 'UNLOADING BUZZER\n(FULL BASKET)' | German: 'ENTLADE-SUMMER (VOLLER KORB)' | France: 'BUZZER DE DÉCHARGEMENT (PANIER PLEIN)' | English: 'UNLOADING BUZZER\n(FULL BASKET)'
  11804 = 'UNLOADING BUZZER \n(OFF IR HEATER)' | English: 'UNLOADING BUZZER \n(OFF IR HEATER)'
  7819 = 'UNLOADING BUZZER \n(SINGLE BASKET)' | German: 'ENTLADE-SUMMER (EINZELNER KORB)' | France: 'BUZZER DE DÉCHARGEMENT (PANIER SIMPLE)' | English: 'UNLOADING BUZZER \n(SINGLE BASKET)'
  6626 = 'UNLOADING FFU UNIT' | German: 'ENTLADEN FFU SICHERUNG' | France: 'DÉCHARGE UNITÉ DE FILTRE' | English: 'UNLOADING FFU UNIT'
  4987 = 'UNLOADING POS 1 COOLING' | English: 'UNLOADING POS 1 COOLING'
  5536 = 'UNLOADING POS 2 COOLING' | English: 'UNLOADING POS 2 COOLING'
  4737 = 'UNLOADING POS 3 COOLING' | English: 'UNLOADING POS 3 COOLING'
  459 = 'UP' | German: 'NACH' | France: 'HAUT' | English: 'UP'
  59 = 'USER' | German: 'BENUTZER' | France: 'UTILISATEUR' | English: 'USER'
  4288 = 'USER\nSETTING' | German: 'BENUTZER\n$SEINSTELLUNGEN' | France: 'PARAMETRES\n$SUTILISATEUR' | English: 'USER\nSETTING'
  3518 = 'USER LEVEL' | German: 'BENUTZEREBENE' | France: 'NIVEAU UTILISATEUR' | English: 'USER LEVEL'
  5968 = 'USER NAME' | German: 'BENUTZERNAME' | France: "NO D'UTILISATEUR" | English: 'USER NAME'
  62 = 'USER SETTING' | German: 'BENUTZER\nEINSTELLUNGEN' | France: 'PARAMETRES\nUTILISATEUR' | English: 'USER SETTING'
  4533 = 'Vaccum' | German: 'VAKUUM' | France: 'SOUS-VIDE' | English: 'Vaccum'
  8785 = 'VACUUM' | German: 'VAKUUM' | France: 'SOUS-VIDE' | English: 'VACUUM'
  6841 = 'VACUUM ABOVE TARGET (kPa)' | German: 'VAKUUM ÜBER SOLLWERT (kPa)' | France: 'SOUS-VIDE AU-DESSUS DE LA CONSIGNE (kPa)' | English: 'VACUUM ABOVE TARGET (kPa)'
  1940 = 'VACUUM ABOVE TARGET kPa' | German: 'VAKUUM ÜBER SOLLWERT kPa' | France: 'SOUS-VIDE AU-DESSUS DE LA CONSIGNE kPa' | English: 'VACUUM ABOVE TARGET kPa'
  6476 = 'VACUUM BELOW TARGET (kPa)' | German: 'VAKUUM UNTER SOLLWERT (kPa)' | France: 'SOUS-VIDE SOUS LA CONSIGNE (kPa)' | English: 'VACUUM BELOW TARGET (kPa)'
  5984 = 'VACUUM BELOW TARGET kPa' | German: 'VAKUUM UNTER SOLLWERT kPa' | France: 'SOUS-VIDE SOUS LA CONSIGNE kPa' | English: 'VACUUM BELOW TARGET kPa'
  4547 = 'VACUUM CALIBRATION' | German: 'VAKUUM KALIBRIERUNG' | France: 'ÉTALONNAGE DU SOUS-VIDE' | English: 'VACUUM CALIBRATION'
  4594 = 'VACUUM LEVEL' | German: 'VAKUUM LEVEL' | France: 'NIVEAU DE SOUS-VIDE' | English: 'VACUUM LEVEL'
  596 = 'VACUUM LEVEL PV ' | German: 'VAKUUM LEVEL PV' | France: 'NIVEAU DE SOUS-VIDE PV' | English: 'VACUUM LEVEL PV '
  6321 = 'VACUUM PRESSURE (bar)' | German: 'VAKUUM DRUCK (bar)' | France: 'PRESSION DE SOUS-VIDE (bar)' | English: 'VACUUM PRESSURE (bar)'
  6778 = 'VACUUM PUMP' | German: 'VAKUUM PUMPE' | France: 'POMPE DE SOUS-VIDE' | English: 'VACUUM PUMP'
  5369 = 'VACUUM PUMP MAJOR SERVICE DAYS' | German: 'VAKUUMPUMPE GROSSE SERVICETAGE' | France: "POMPE DE SOUS-VIDE GRANDES JOURNÉES D'ENTRETIEN" | English: 'VACUUM PUMP MAJOR SERVICE DAYS'
  4691 = 'VACUUM PUMP ROUTINE SERVICE DAYS' | German: 'VAKUUMPUMPE ROUTINEWARTUNGSTAGE' | France: 'POMPE DE SOUS-VIDE JOURS DE MAINTENANCE DE ROUTINE' | English: 'VACUUM PUMP ROUTINE SERVICE DAYS'
  1822 = 'VACUUM PUMP RUN TIMER' | German: 'VAKUUMPUMPEN-LAUFZEITMESSER' | France: 'COMPTEUR DE TEMPS DE LA POMPE À SOUS-VIDE' | English: 'VACUUM PUMP RUN TIMER'
  853 = 'VACUUM PUMP SERVICE DAYS' | German: 'VAKUUMPUMPEN-WARTUNGSTAGE' | France: "JOURS D'ENTRETIEN DE LA POMPE À SOUS-VIDE" | English: 'VACUUM PUMP SERVICE DAYS'
  3013 = 'VACUUM PUMP SERVICE DAYs' | German: 'VAKUUMPUMPEN-WARTUNGSTAGE' | France: "JOURS D'ENTRETIEN DE LA POMPE À SOUS-VIDE" | English: 'VACUUM PUMP SERVICE DAYs'
  1935 = 'VACUUM PUMP SERVICE HOUR' | German: 'VAKUUMPUMPE SERVICE STUNDE' | France: 'POMPE À SOUS-VIDE HEURE DE SERVICE' | English: 'VACUUM PUMP SERVICE HOUR'
  2670 = 'VACUUM PUMP SERVICE ROUTINE' | German: 'VAKUUMPUMPE SERVICE ROUTINE' | France: 'POMPE À SOUS-VIDE DE SERVICE ROUTINE' | English: 'VACUUM PUMP SERVICE ROUTINE'
  6275 = 'VACUUM PUMP TIMER' | German: 'VAKUUMPUMPE TIMER' | France: 'POMPE À SOUS-VIDE MINUTERIE' | English: 'VACUUM PUMP TIMER'
  1450 = 'VACUUM SYSTEM' | German: 'VAKUUMSYSTEM' | France: 'SYSTÈME DE SOUS-VIDE' | English: 'VACUUM SYSTEM'
  7519 = 'VACUUM SYSTEM (kpa)' | German: 'VAKUUMSYSTEM (kpa)' | France: 'SYSTÈME DE SOUS-VIDE (kpa)' | English: 'VACUUM SYSTEM (kpa)'
  3009 = 'VELOCITY (mm/s)' | German: 'GESCHWINDIGKEIT (mm/s)' | France: 'VITESSE (mm/s)' | English: 'VELOCITY (mm/s)'
  1563 = 'VERTICAL' | German: 'VERTIKAL' | France: 'VERTICALE' | English: 'VERTICAL'
  4494 = 'VOLUME PER BASKET (ml)' | German: 'VOLUMEN PER KORB (ml)' | France: 'VOLUME PAR PANIER(ml)' | English: 'VOLUME PER BASKET (ml)'
  2338 = 'WASHING' | German: 'Washen' | France: 'LAVAGE' | English: 'WASHING'
  2654 = 'WEDNESDAY' | German: 'Mittwoch' | France: 'Mercredi' | English: 'WEDNESDAY'
  2581 = 'Write Done' | German: 'SCHREIBEN ERLEDIGT' | France: 'ÉCRIRE FAIT' | English: 'Write Done'
  4553 = 'μS' | German: 'μS' | France: 'μS' | English: 'μS'
END_TEXTLIST

// ---- VISUs/IO MONITORING/IO_Monitoring.TcVIS
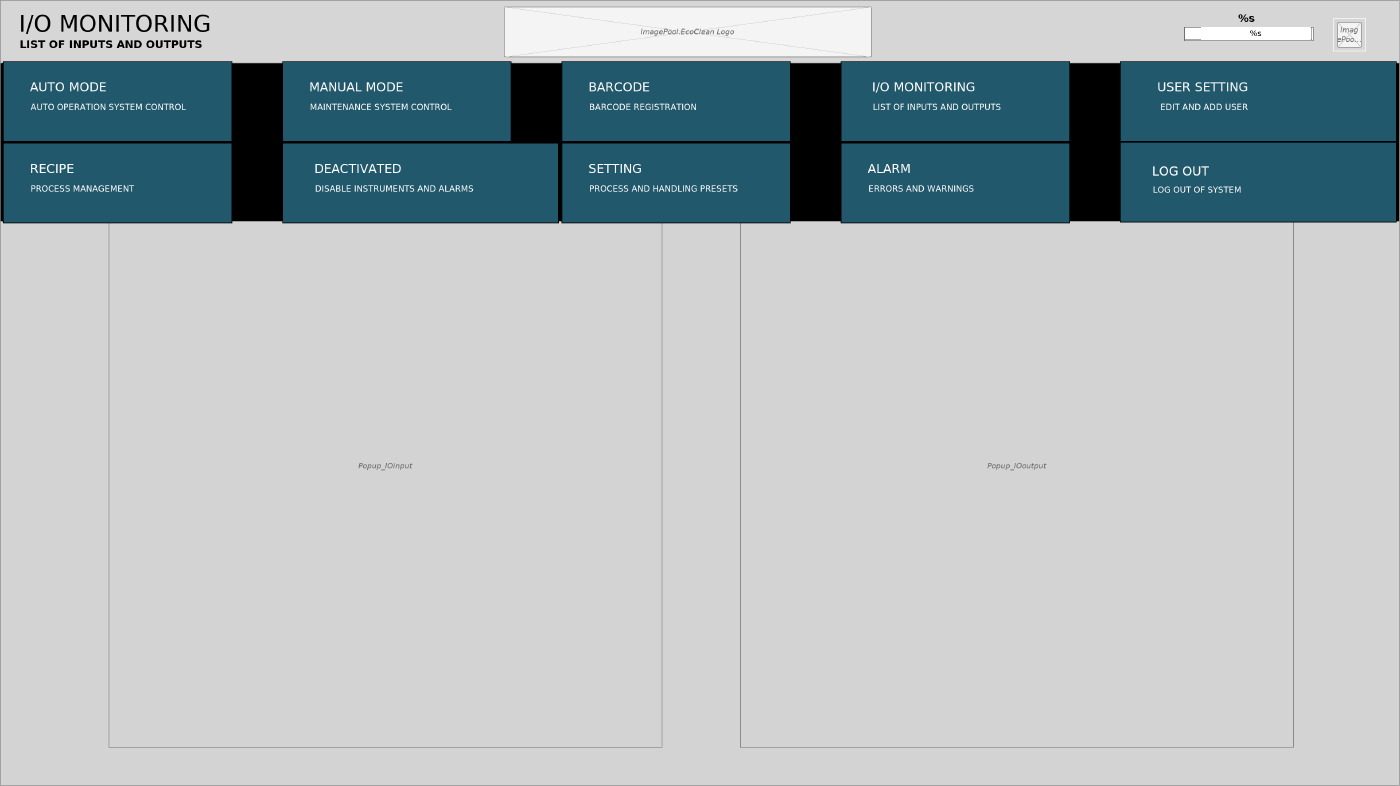
VISUALIZATION IO_Monitoring  // 1920x1079
    Rectangle (0,98 1920x981)
    Group (141,247 1639x790)
        Rectangle (0,0 774x790)
        Rectangle (865,0 774x790)
    Rectangle (0,63 1920x26)
        p3528305787: HMI_Ctrl.ANIMATION3
    Rectangle (0,0 1919x85)
    Label (23,6 310x53), "I/O MONITORING"
    Label (24,49 320x24), "LIST OF INPUTS AND OUTPUTS"
    Group (1828,25 45x45)
        OnMouseClick: toggle HMI_Ctrl.MenuButton
        RoundedRectangle (0,0 45x45), colour toggle: HMI_Ctrl.MenuButton
        Image (6,5 33x35), image: ImagePool.Menu Button
    Frame (149,253 759x773)
        shows Popup_IOinput()
    Frame (1015,253 759x773)
        shows Popup_IOoutput()
    Image (691,9 504x69), image: ImagePool.EcoClean Logo
    Group (1621,14 180x42)
        Rectangle (0,0 177x22), "%s", text variable: DSLocalSystemTimeML.sCurrentDT24Hr_General
        Button (3,23 177x19), image: VisuSymbols.Symbols.AddUser
        Rectangle (26,23 150x18), "%s", text variable: fbHmiTF1800_UserlevelManagement.dsHmiUserStatus_Active.sLoginName
    Label (419,195 125x53), "INPUT"
    Label (1324,195 153x53), "OUTPUT"
    Frame (0,84 1918x221), invisible if: HMI_Ctrl.CloseMenuButton
        shows Popup_MenuPage()
END_VISUALIZATION

// ---- VISUs/MANUAL/Manual_AllStation.TcVIS
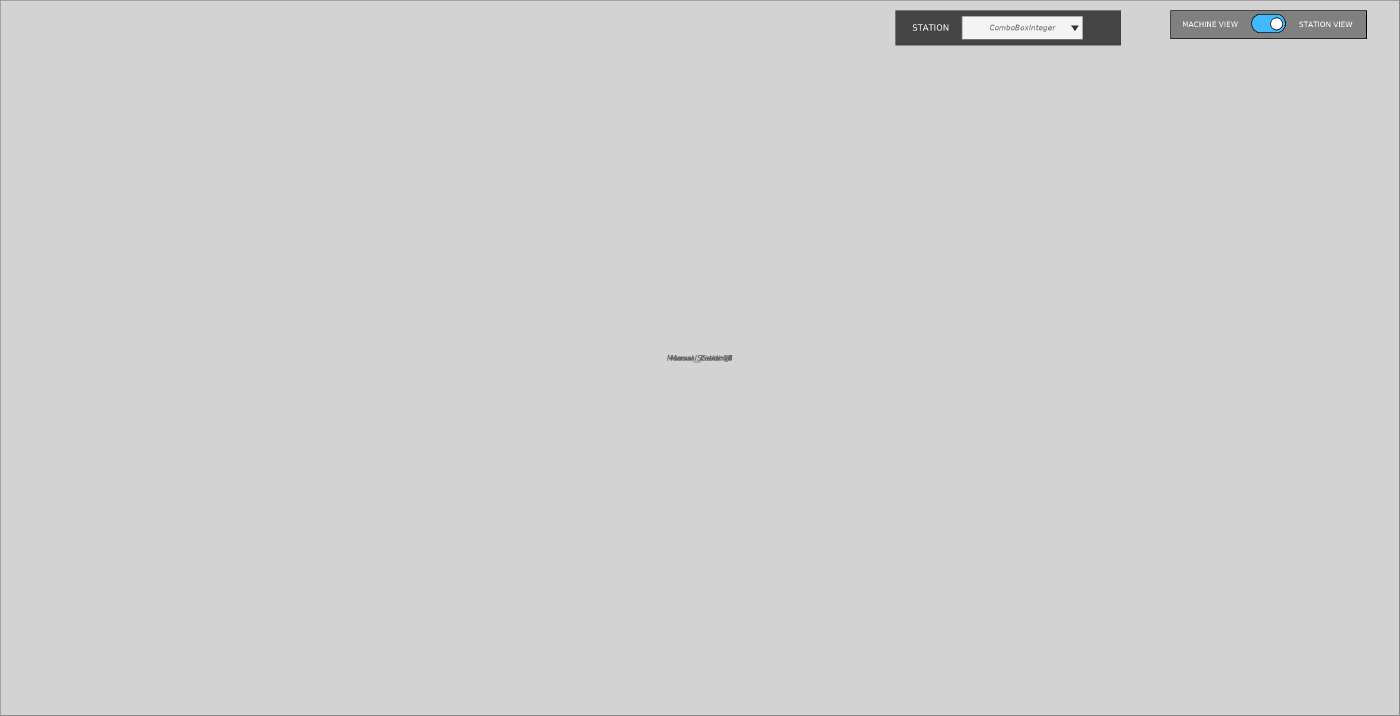
VISUALIZATION Manual_AllStation  // 1920x983
    Rectangle (0,0 1920x983)
    Frame (0,0 1920x983), invisible if: HMI_Ctrl.StationInfoPageNo <> 1
        shows Manual_Station01()
    Frame (0,0 1920x983), invisible if: HMI_Ctrl.StationInfoPageNo <> 2
        shows Manual_Station02()
    Frame (0,0 1920x983), invisible if: HMI_Ctrl.StationInfoPageNo <> 3
        shows Manual_Station03()
    Frame (0,0 1920x983), invisible if: HMI_Ctrl.StationInfoPageNo <> 4
        shows Manual_Station04()
    Frame (0,0 1920x983), invisible if: HMI_Ctrl.StationInfoPageNo <> 5
        shows Manual_Station05()
    Frame (0,0 1920x983), invisible if: HMI_Ctrl.StationInfoPageNo <> 6
        shows Manual_Station06()
    Frame (0,0 1920x983), invisible if: HMI_Ctrl.StationInfoPageNo <> 7
        shows Manual_Loading()
    Frame (0,0 1920x983), invisible if: HMI_Ctrl.StationInfoPageNo <> 0
        shows Manual_General()
    Group (1605,13 269x41)
        RoundedRectangle (0,1 269x39)
        Label (1,0 108x41), "MACHINE VIEW"
        Label (161,0 105x41), "STATION VIEW"
        Group (111,6 47x26)
            OnMouseClick: toggle HMI_Ctrl.AutoStationViewEnable
            Ellipse (0,0 26x26)
            Ellipse (21,0 26x26)
            RoundedRectangle (8,0 29x26)
            Ellipse (1,1 24x24)
            Ellipse (23,1 23x24)
            RoundedRectangle (9,1 28x24)
            Ellipse (26,5 17x17)
    Group (1228,14 272x48)
        RoundedRectangle (0,0 309x48)
        Label (20,12 79x24), "STATION"
    ComboBoxInteger (1319,22 166x32), variable: HMI_Ctrl.StationInfoPageNo, invisible if: NOT HMI_Ctrl.AutoStationViewEnable, text list: 'TextList_ManualPage'
END_VISUALIZATION

// ---- VISUs/MANUAL/Manual_Page.TcVIS
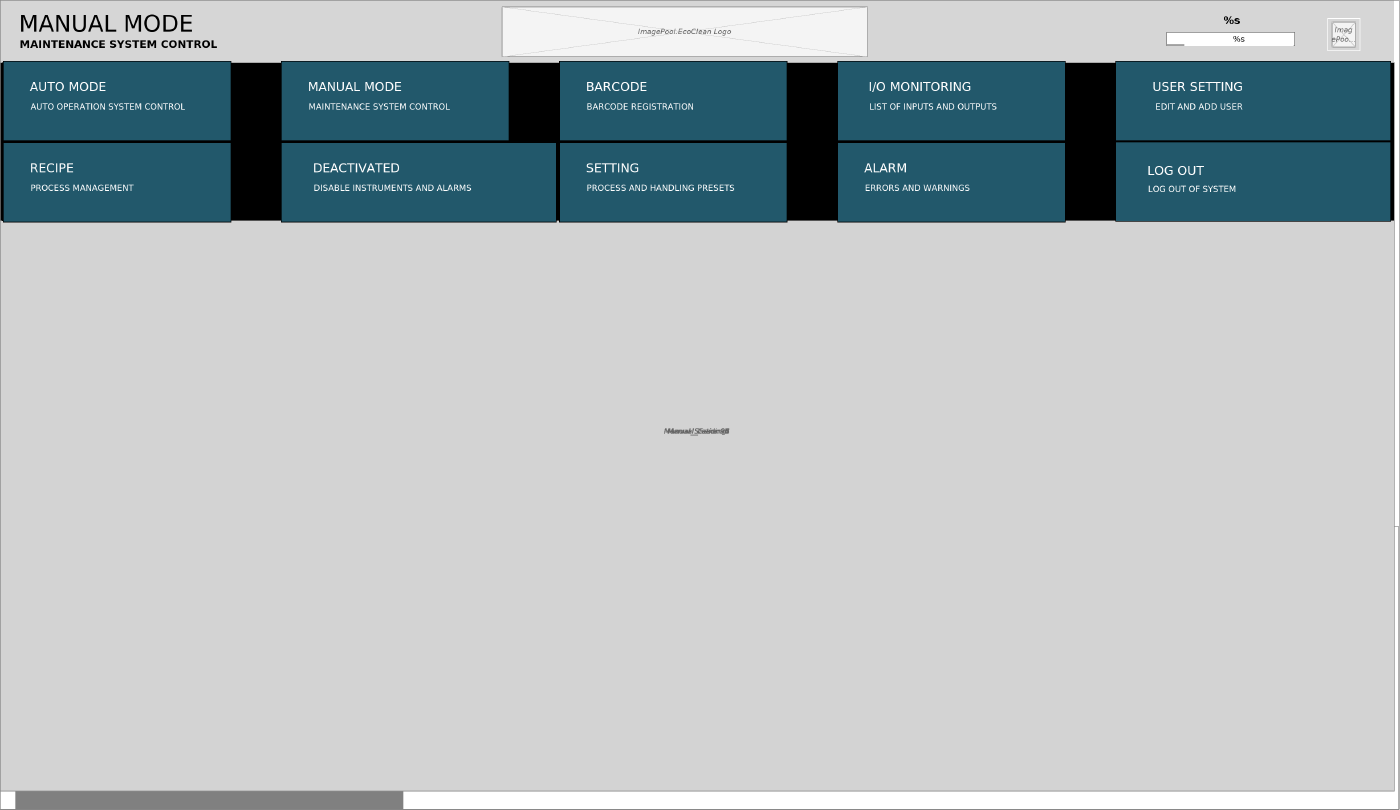
VISUALIZATION Manual_Page  // 1928x1116
    Rectangle (0,88 1919x985)
    Rectangle (1356,531 562x27)
    Rectangle (1356,558 562x143)
    Rectangle (2,431 606x270)
    Rectangle (2,135 606x267)
    Rectangle (2,703 1915x27)
    Rectangle (2,404 607x27)
    Rectangle (610,531 746x27)
    Rectangle (610,558 744x143)
    Rectangle (0,63 1920x26)
        p3528305787: HMI_Ctrl.ANIMATION3
    Rectangle (0,0 1919x85)
    Label (23,6 564x53), "MANUAL MODE"
    Label (24,49 541x24), "MAINTENANCE SYSTEM CONTROL"
    Group (1828,25 45x45)
        OnMouseClick: toggle HMI_Ctrl.MenuButton
        RoundedRectangle (0,0 45x45), colour toggle: HMI_Ctrl.MenuButton
        Image (6,5 33x35), image: ImagePool.Menu Button
    Frame (614,124 1281x394)
        shows Popup_Machine_Manual()
    Group (20,144 357x87)
        Group (0,0 144x27)
            Rectangle (0,0 144x27)
            Label (14,2 56x24), "ARM"
        Group (6,43 100x43)
            RoundedRectangle (0,0 100x6), colour toggle: ARbArmVertHomeDone[1]
            Rectangle (0,11 100x32), "VERTICAL", colour toggle: bArm1VertHomeStart_30
                toggle bArm1VertHomeStart_30
        Group (130,44 101x43)
            RoundedRectangle (1,0 100x6), colour toggle: ARDSArmCtrl[1].AR3sbPositionCfm[2,1,1]
            Rectangle (0,11 100x32), "UP", colour toggle: bArm1VertLD1Up_30
                toggle bArm1VertLD1Up_30
        Group (257,44 100x43)
            RoundedRectangle (0,0 100x6), colour toggle: ARbArmHorzHomeDone[1]
            Rectangle (0,11 100x32), "HORIZONTAL", colour toggle: bArm1HorzHomeStart_30
                toggle bArm1HorzHomeStart_30
    Group (405,355 188x28)
        Label (0,2 112x24), "ARM HOMING :"
        Rectangle (114,0 74x28), "Reset", colour toggle: bArmHomeResetbit
            tap bArmHomeResetbit
    Label (659,569 110x24), "ARM POSITION"
    Label (1169,569 110x24), "PRODUCT INFO"
    Label (1171,602 82x24), "RECIPE NO."
    Label (1171,630 63x24), "QUALITY"
    Rectangle (1248,606 100x17), "%i", text variable: DSArmBasketInfo[1].iProductRecipeNo
        OnMouseDown: write the text variable via VisuDialogs.Numpad, min 0, max 40
    Rectangle (1248,634 100x17), "%s", text variable: DSArmBasketInfo[1].sProductQuality
    Image (691,9 504x69), image: ImagePool.EcoClean Logo
    Frame (-2,725 1928x391)
        shows Popup_ArmControl()
    Label (856,704 143x24), "ARM CONTROL"
    Rectangle (742,634 150x17), "%0.01f", text variable: DSArm1HorzConfig.lrGen_Out_CurrentPos
    Label (638,602 82x24), "VERTICAL"
    Label (638,630 97x24), "HORIZONTAL"
    Rectangle (742,606 150x17), "%0.01f", text variable: DSArm1VertConfig.lrGen_Out_CurrentPos
    Label (908,535 133x24), "ARM INFO"
    Group (43,442 249x248)
        Ellipse (0,0 249x248)
        RoundedRectangle (90,12 70x223)
        RoundedRectangle (13,89 224x69)
        RoundedRectangle (89,88 73x72)
        Group (92,163 70x69)
            tap ARbArmVertJogFwd[1]
            PushSwitch (0,0 70x69), variable: ARbArmVertJogFwd[1], behaviour: TOGGLE, style: Switch-PushSwitch-Blue
            Image (14,17 40x40), image: VisuSymbols.Symbols.TriangleDown
        Group (17,89 70x69)
            tap ARbArmHorzJogRwd[1]
            PushSwitch (0,0 70x69), variable: ARbArmHorzJogRwd[1], behaviour: TOGGLE, style: Switch-PushSwitch-Blue
            Image (10,14 40x40), image: VisuSymbols.Symbols.TriangleLeft
        Group (165,89 70x69)
            tap ARbArmHorzJogFwd[1]
            PushSwitch (0,0 70x69), variable: ARbArmHorzJogFwd[1], behaviour: TOGGLE, style: Switch-PushSwitch-Blue
            Image (17,14 40x40), image: VisuSymbols.Symbols.TriangleRight
        Group (91,17 70x69)
            tap ARbArmVertJogRwd[1]
            PushSwitch (0,0 70x69), variable: ARbArmVertJogRwd[1], behaviour: TOGGLE, style: Switch-PushSwitch-Blue
            Image (15,11 40x40), image: VisuSymbols.Symbols.TriangleUp
    Rectangle (303,547 220x27)
    Label (329,550 157x24), "ARM JOG VELO (mm/s)"
    Label (310,587 82x24), "VERTICAL"
    Label (310,618 97x24), "HORIZONTAL"
    Rectangle (420,592 120x17), "%0.01f", text variable: ARrArmVertJogPercent[1]
        OnMouseDown: write the text variable via VisuDialogs.Numpad, min 2, max 100
    Rectangle (420,623 121x17), "%0.01f", text variable: ARrArmHorzJogPercent[1]
        OnMouseDown: write the text variable via VisuDialogs.Numpad, min 2, max 100
    Label (410,618 13x24), ":"
    Label (410,588 13x24), ":"
    Rectangle (2,108 607x27)
    Label (226,110 147x24), "HOMING SECTION"
    Label (215,407 97x24), "JOG MODE"
    Group (9,437 569x260), invisible if: bArmJogEnable
        Rectangle (0,0 525x255), invisible if: bArmJogEnable
        Label (184,94 173x59), "N/A", invisible if: bArmJogEnable
    Group (21,741 1876x333)
        Rectangle (0,0 534x610), invisible if: bArmHomingComplete[1]
        Label (199,194 138x170), "N/A", invisible if: bArmHomingComplete[1]
    Rectangle (495,404 98x26), "ENABLE", colour toggle: bArmJogEnable
        toggle bArmJogEnable
    Group (1603,103 269x41), invisible if: HMI_Ctrl.AutoStationViewEnable
        RoundedRectangle (0,1 269x39)
        Label (1,0 108x41), "MACHINE VIEW"
        Label (161,0 105x41), "STATION VIEW"
        Group (111,6 47x26)
            OnMouseClick: toggle HMI_Ctrl.AutoStationViewEnable
            Group (0,0 47x26)
                Ellipse (0,0 26x26)
                Ellipse (21,0 26x26)
                RoundedRectangle (8,0 29x26)
            Ellipse (1,1 24x24)
            Ellipse (23,1 23x24)
            RoundedRectangle (9,1 28x24)
            Ellipse (5,5 17x17)
    Group (1606,17 179x46)
        Button (0,27 177x19), image: VisuSymbols.Symbols.AddUser
        Rectangle (25,28 150x18), "%s", text variable: fbHmiTF1800_UserlevelManagement.dsHmiUserStatus_Active.sLoginName
        Rectangle (2,0 177x22), "%s", text variable: DSLocalSystemTimeML.sCurrentDT24Hr_General
    Label (1558,534 196x24), "MANUAL BASKET LOAD"
    Label (1437,632 127x24), "RECIPE NAME"
    Label (1429,569 110x24), "PRODUCT INFO"
    Label (1441,602 82x24), "RECIPE NO."
    Rectangle (1538,634 349x17), "%s", text variable: ARsProductRecipeDescription[iUserDefineProductRecipeNo]
    Rectangle (1538,606 100x17), "%i", text variable: iUserDefineProductRecipeNo
        OnMouseDown: write the text variable via VisuDialogs.Numpad, min 0, max 40
    Frame (0,98 1920x992), invisible if: NOT HMI_Ctrl.AutoStationViewEnable
        shows Manual_AllStation()
    Frame (0,84 1918x221), invisible if: HMI_Ctrl.CloseMenuButton
        shows Popup_MenuPage()
END_VISUALIZATION

// ---- VISUs/POPUP/Manual_Exit_Popup.TcVIS
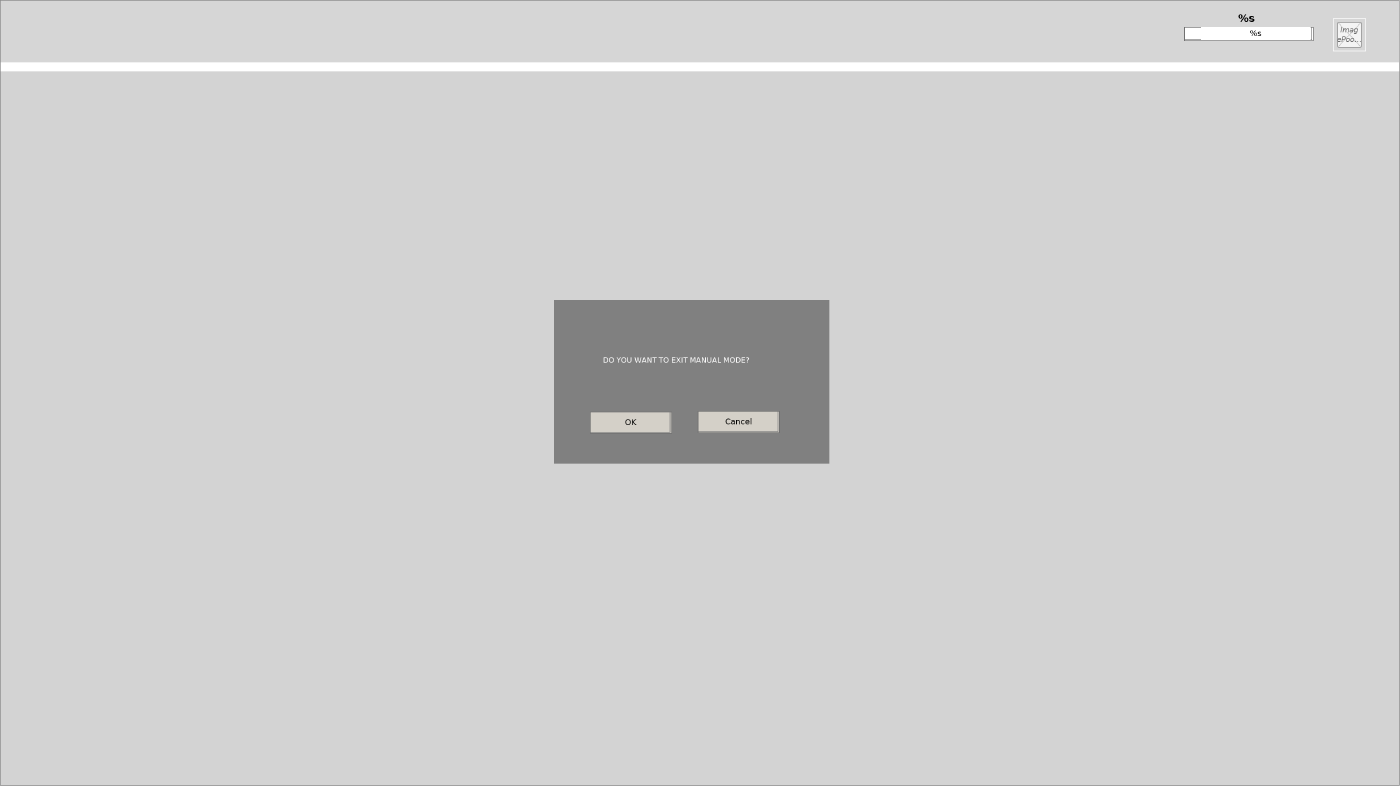
VISUALIZATION Manual_Exit_Popup  // 1920x1079
    Rectangle (0,98 1920x981)
    Rectangle (0,63 1920x26)
        p3528305787: HMI_Ctrl.ANIMATION3
    Rectangle (0,0 1919x85)
    Group (1828,25 45x45)
        OnMouseClick: toggle HMI_Ctrl.MenuButton
        RoundedRectangle (0,0 45x45), colour toggle: HMI_Ctrl.MenuButton
        Image (6,5 33x35), image: ImagePool.Menu Button
    Rectangle (760,412 377x224)
    Label (809,413 209x24)
    Label (824,469 241x51), "DO YOU WANT TO EXIT MANUAL MODE?"
    Button (809,565 112x30), "OK"
        tap bManualExitConfirm
    Button (957,564 112x30), "Cancel"
        tap bManualExitCancel
    Group (1621,14 180x42)
        Rectangle (0,0 177x22), "%s", text variable: DSLocalSystemTimeML.sCurrentDT24Hr_General
        Button (3,23 177x19), image: VisuSymbols.Symbols.AddUser
        Rectangle (26,23 150x18), "%s", text variable: fbHmiTF1800_UserlevelManagement.dsHmiUserStatus_Active.sLoginName
END_VISUALIZATION

// ---- VISUs/POPUP/Popup_Parameter.TcVIS
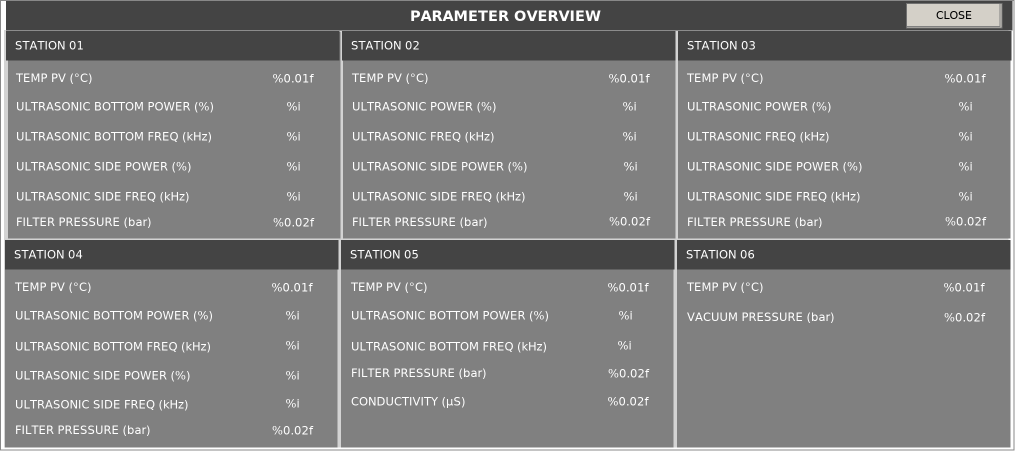
VISUALIZATION Popup_Parameter  // 1015x451
    Rectangle (4,30 1004x417)
    Rectangle (6,1 1006x29)
    Label (407,4 216x24), "PARAMETER OVERVIEW"
    Button (906,3 96x25), "CLOSE"
        OnMouseDown: execute { bParameterPopupPageOn:=0; }
    Rectangle (677,241 333x206)
    Rectangle (677,240 333x29)
    Label (683,242 96x25), "STATION 06"
    Label (684,267 199x40), "TEMP PV (°C)"
    Rectangle (921,264 86x47), "%0.01f", text variable: ARrStnTempPV[6]
    Label (684,296 200x42), "VACUUM PRESSURE (bar)"
    Rectangle (920,297 89x41), "%0.02f", text variable: ARrStnVacuumPV[6]
    Rectangle (8,32 332x206)
    Rectangle (6,31 333x29)
    Label (12,33 96x25), "STATION 01"
    Label (13,58 199x40), "TEMP PV (°C)"
    Rectangle (250,55 86x47), "%0.01f", text variable: ARrStnTempPV[1]
    Label (13,94 235x25), "ULTRASONIC BOTTOM POWER (%)"
    Rectangle (253,93 81x27), "%i", text variable: ARiStnUSBtmAPv[1]
    Label (13,201 163x42), "FILTER PRESSURE (bar)"
    Rectangle (249,202 89x41), "%0.02f", text variable: ARrStnFilterPressurePV[1]
    Label (13,123 240x27), "ULTRASONIC BOTTOM FREQ (kHz)"
    Rectangle (244,117 99x39), "%i", text variable: ARiStnUSBtmAFreqPv[1]
    Label (13,183 240x27), "ULTRASONIC SIDE FREQ (kHz)"
    Label (13,154 235x25), "ULTRASONIC SIDE POWER (%)"
    Rectangle (253,153 81x27), "%i", text variable: ARiStnUSSideAPv[1]
    Rectangle (244,177 99x39), "%i", text variable: ARiStnUSSideAFreqPv[1]
    Rectangle (343,32 332x206)
    Rectangle (342,31 333x29)
    Label (348,33 96x25), "STATION 02"
    Label (349,58 199x40), "TEMP PV (°C)"
    Rectangle (586,55 86x47), "%0.01f", text variable: ARrStnTempPV[2]
    Label (349,94 303x25), "ULTRASONIC POWER (%)"
    Rectangle (589,93 81x27), "%i", text variable: ARiStnUSBtmAPv[2]
    Label (349,201 169x42), "FILTER PRESSURE (bar)"
    Rectangle (585,201 89x41), "%0.02f", text variable: ARrStnFilterPressurePV[2]
    Label (349,123 231x27), "ULTRASONIC FREQ (kHz)"
    Rectangle (580,117 99x39), "%i", text variable: ARiStnUSBtmAFreqPv[2]
    Label (349,154 235x25), "ULTRASONIC SIDE POWER (%)"
    Label (349,183 240x27), "ULTRASONIC SIDE FREQ (kHz)"
    Rectangle (590,153 81x27), "%i", text variable: ARiStnUSSideAPv[2]
    Rectangle (581,177 99x39), "%i", text variable: ARiStnUSSideAFreqPv[2]
    Group (678,31 337x212)
        Rectangle (0,1 332x206)
        Rectangle (0,0 333x29)
        Label (6,2 96x25), "STATION 03"
        Label (6,27 199x40), "TEMP PV (°C)"
        Rectangle (244,24 86x47), "%0.01f", text variable: ARrStnTempPV[3]
        Rectangle (247,62 81x27), "%i", text variable: ARiStnUSBtmAPv[3]
        Label (6,170 165x42), "FILTER PRESSURE (bar)"
        Rectangle (243,170 89x41), "%0.02f", text variable: ARrStnFilterPressurePV[3]
        Label (6,63 173x25), "ULTRASONIC POWER (%)"
        Label (6,92 164x27), "ULTRASONIC FREQ (kHz)"
        Rectangle (238,86 99x39), "%i", text variable: ARiStnUSBtmAFreqPv[3]
        Label (6,123 235x25), "ULTRASONIC SIDE POWER (%)"
        Label (6,152 240x27), "ULTRASONIC SIDE FREQ (kHz)"
        Rectangle (247,122 81x27), "%i", text variable: ARiStnUSSideAPv[1]
        Rectangle (238,146 99x39), "%i", text variable: ARiStnUSSideAFreqPv[1]
    Label (12,332 376x27), "ULTRASONIC FREQ (kHz)"
    Rectangle (5,241 332x206)
    Rectangle (5,240 333x29)
    Label (11,242 96x25), "STATION 04"
    Label (12,267 199x40), "TEMP PV (°C)"
    Rectangle (249,264 86x47), "%0.01f", text variable: ARrStnTempPV[4]
    Label (12,303 232x25), "ULTRASONIC BOTTOM POWER (%)"
    Rectangle (252,302 81x27), "%i", text variable: ARiStnUSBtmAPv[4]
    Label (12,409 170x42), "FILTER PRESSURE (bar)"
    Rectangle (248,410 89x41), "%0.02f", text variable: ARrStnFilterPressurePV[4]
    Rectangle (243,326 99x39), "%i", text variable: ARiStnUSBtmAFreqPv[4]
    Label (12,333 182x27), "ULTRASONIC BOTTOM FREQ (kHz)"
    Label (12,363 201x25), "ULTRASONIC SIDE POWER (%)"
    Rectangle (252,362 81x27), "%i", text variable: ARiStnUSSideAPv[4]
    Rectangle (243,384 99x39), "%i", text variable: ARiStnUSSideAFreqPv[4]
    Label (12,391 210x27), "ULTRASONIC SIDE FREQ (kHz)"
    Group (341,240 341x207)
        Rectangle (0,1 332x206)
        Rectangle (0,0 333x29)
        Label (6,2 96x25), "STATION 05"
        Label (7,27 199x40), "TEMP PV (°C)"
        Rectangle (244,24 86x47), "%0.01f", text variable: ARrStnTempPV[5]
        Label (7,112 165x42), "FILTER PRESSURE (bar)"
        Rectangle (243,113 89x41), "%0.02f", text variable: ARrStnFilterPressurePV[5]
        Label (7,149 173x25), "CONDUCTIVITY (μS)"
        Rectangle (233,152 108x19), "%0.02f", text variable: ARrStnConductivityPV[5]
        Label (7,63 228x25), "ULTRASONIC BOTTOM POWER (%)"
        Rectangle (244,62 81x27), "%i", text variable: ARiStnUSBtmAPv[5]
        Rectangle (234,86 99x39), "%i", text variable: ARiStnUSBtmAFreqPv[5]
        Label (7,93 223x27), "ULTRASONIC BOTTOM FREQ (kHz)"
END_VISUALIZATION

// ---- VISUs/POPUP/Popup_Parameter_Saved.TcVIS
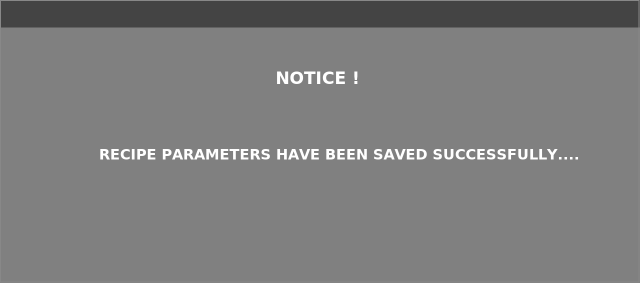
VISUALIZATION Popup_Parameter_Saved  // 640x283
    Rectangle (0,0 640x283)
    Rectangle (1,0 639x27)
    Label (262,66 101x24), "NOTICE !"
    Label (96,100 516x109), "RECIPE PARAMETERS HAVE BEEN SAVED SUCCESSFULLY...."
END_VISUALIZATION

// ---- VISUs/POPUP/Vacuum_Calibration.TcVIS
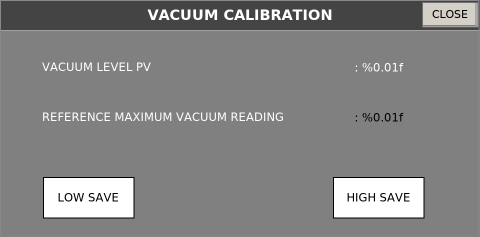
VISUALIZATION Vacuum_Calibration  // 480x237
    Rectangle (0,31 480x206)
    Rectangle (0,0 480x30), "VACUUM CALIBRATION"
    Label (39,47 129x40), "VACUUM LEVEL PV"
    Rectangle (336,44 86x47), ": %0.01f", text variable: ARrStnVacuumPV[6]
    Label (39,97 285x40), "REFERENCE MAXIMUM VACUUM READING"
    Rectangle (336,94 86x47), ": %0.01f", text variable: ARlrStnVacuumMaxReadSV[6]
        OnMouseDown: write the text variable via VisuDialogs.Numpad
    Rectangle (43,177 91x41), "LOW SAVE", colour toggle: ARbStnLowVacuumLvlSave[6]
        tap ARbStnLowVacuumLvlSave[6]
    Rectangle (333,177 91x41), "HIGH SAVE", colour toggle: ARbStnHighVacuumLvlSave[6]
        tap ARbStnHighVacuumLvlSave[6]
    Button (422,2 56x25), "CLOSE"
        toggle bManualCalibratePageOn
END_VISUALIZATION

// ---- VISUs/Popup_Machine.TcVIS
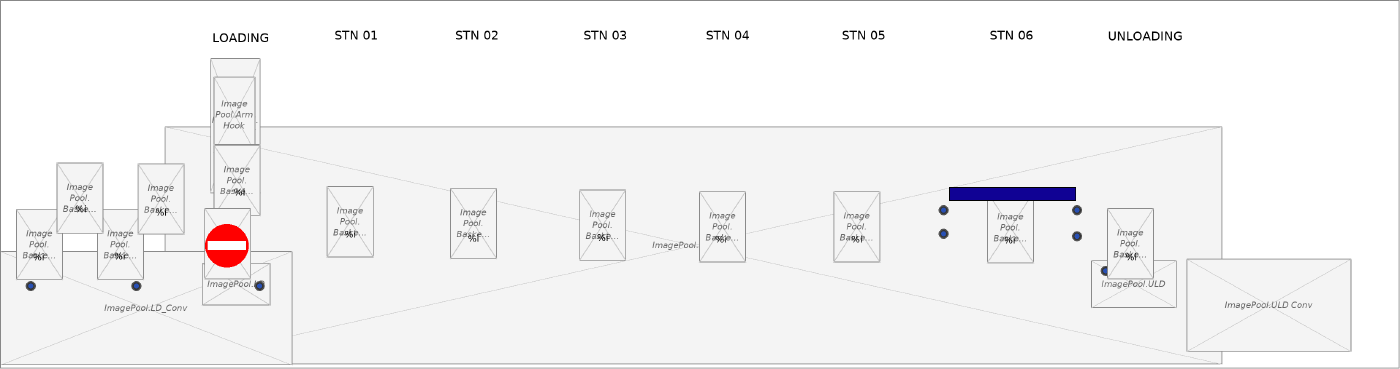
VISUALIZATION Popup_Machine  // 1658x438
    Rectangle (0,0 1658x438)
    Image (195,150 1252x282), image: ImagePool.Machine
    Label (379,22 86x40), "STN 01"
    Label (522,22 86x40), "STN 02"
    Label (674,22 86x40), "STN 03"
    Label (819,22 86x40), "STN 04"
    Label (980,22 86x40), "STN 05"
    Label (1155,22 86x40), "STN 06"
    Label (232,22 106x46), "LOADING"
    Label (1294,22 125x42), "UNLOADING"
    Image (0,298 346x135), image: ImagePool.LD_Conv
    Image (239,312 81x50), image: ImagePool.LD
    Image (249,69 59x160), image: ImagePool.Arm Body
        p3560616238: HMI_Function.MotionX
    Image (253,91 49x90), image: ImagePool.Arm Hook
        p3560616238: HMI_Function.MotionX
        p2738717112: HMI_Function.MotionY
    Image (1405,307 195x110), image: ImagePool.ULD Conv
    Image (1292,309 101x56), image: ImagePool.ULD
    Lamp1 (301,333 13x13), variable: ARbDI[eX13002_LoadingConveyorSensor_Pick], style: Lamp-Lamp1-Blue
    Lamp1 (1303,315 13x13), variable: ARbDI[eX12011_UnloadingSensor_BasketDetection], style: Lamp-Lamp1-Blue
    Image (387,221 55x84), invisible if: NOT.ARbBasketBdFlag[2], image: ImagePool.Basket Red
    Rectangle (399,261 32x31), "%i", text variable: DSStnBasketInfo[1].iProductRecipeNo, invisible if: NOT.ARbBasketBdFlag[2]
    Group (387,221 55x84)
        Image (0,0 55x84), invisible if: NOT.ARbBasketGdFlag[2], image: ImagePool.Basket Green
        Rectangle (12,42 32x31), "%i", text variable: DSStnBasketInfo[1].iProductRecipeNo, invisible if: NOT.ARbBasketGdFlag[2]
    Group (533,223 55x84)
        Image (0,0 55x84), invisible if: NOT.ARbBasketBdFlag[3], image: ImagePool.Basket Red
        Rectangle (11,44 32x31), "%i", text variable: DSStnBasketInfo[2].iProductRecipeNo, invisible if: NOT.ARbBasketBdFlag[3]
    Group (533,223 55x84)
        Image (0,0 55x84), invisible if: NOT.ARbBasketGdFlag[3], image: ImagePool.Basket Green
        Rectangle (12,45 32x31), "%i", text variable: DSStnBasketInfo[2].iProductRecipeNo, invisible if: NOT.ARbBasketGdFlag[3]
    Image (686,225 55x84), invisible if: NOT.ARbBasketBdFlag[4], image: ImagePool.Basket Red
    Rectangle (698,268 32x31), "%i", text variable: DSStnBasketInfo[3].iProductRecipeNo, invisible if: NOT.ARbBasketBdFlag[4]
    Group (686,225 55x84)
        Image (0,0 55x84), invisible if: NOT.ARbBasketGdFlag[4], image: ImagePool.Basket Green
        Rectangle (12,42 32x31), "%i", text variable: DSStnBasketInfo[3].iProductRecipeNo, invisible if: NOT.ARbBasketGdFlag[4]
    Group (828,227 55x84)
        Image (0,0 55x84), invisible if: NOT.ARbBasketBdFlag[5], image: ImagePool.Basket Red
        Rectangle (12,43 32x31), "%i", text variable: DSStnBasketInfo[4].iProductRecipeNo, invisible if: NOT.ARbBasketBdFlag[5]
    Group (828,227 55x84)
        Image (0,0 55x84), invisible if: NOT.ARbBasketGdFlag[5], image: ImagePool.Basket Green
        Rectangle (10,42 32x31), "%i", text variable: DSStnBasketInfo[4].iProductRecipeNo, invisible if: NOT.ARbBasketGdFlag[5]
    Group (987,227 55x84)
        Image (0,0 55x84), invisible if: NOT.ARbBasketBdFlag[6], image: ImagePool.Basket Red
        Rectangle (12,43 32x31), "%i", text variable: DSStnBasketInfo[5].iProductRecipeNo, invisible if: NOT.ARbBasketBdFlag[6]
    Group (987,227 55x84)
        Image (0,0 55x84), invisible if: NOT.ARbBasketGdFlag[6], image: ImagePool.Basket Green
        Rectangle (12,42 32x31), "%i", text variable: DSStnBasketInfo[5].iProductRecipeNo, invisible if: NOT.ARbBasketGdFlag[6]
    Group (1169,228 55x84)
        Image (0,0 55x84), invisible if: NOT.ARbBasketBdFlag[7], image: ImagePool.Basket Red
        Rectangle (13,42 32x31), "%i", text variable: DSStnBasketInfo[6].iProductRecipeNo, invisible if: NOT.ARbBasketBdFlag[7]
    Group (1169,228 55x84)
        Image (0,0 55x84), invisible if: NOT.ARbBasketGdFlag[7], image: ImagePool.Basket Green
        Rectangle (11,42 32x31), "%i", text variable: DSStnBasketInfo[6].iProductRecipeNo, invisible if: NOT.ARbBasketGdFlag[7]
    Group (1311,247 55x84)
        Image (0,0 55x84), invisible if: NOT.ARbBasketBdFlag[12], image: ImagePool.Basket Red
        Rectangle (12,42 32x31), "%i", text variable: AR2sDSCv_UldConfirmBasketInfo[1,1].iProductRecipeNo, invisible if: NOT.ARbBasketBdFlag[12]
    Group (1311,247 55x84)
        Image (0,0 55x84), invisible if: NOT.ARbBasketGdFlag[12], image: ImagePool.Basket Green
        Rectangle (13,43 32x31), "%i", text variable: AR2sDSCv_UldConfirmBasketInfo[1,1].iProductRecipeNo, invisible if: NOT.ARbBasketGdFlag[12]
    Image (253,171 55x84), invisible if: NOT.ARbBasketBdFlag[16], image: ImagePool.Basket Red
        p2738717112: HMI_Function.MotionY
        p3560616238: HMI_Function.MotionX
    Rectangle (269,214 32x31), "%i", text variable: DSArmBasketInfo[1].iProductRecipeNo, invisible if: NOT.ARbBasketBdFlag[16]
        p3560616238: HMI_Function.MotionX
        p2738717112: HMI_Function.MotionY
    Image (253,172 55x84), invisible if: NOT.ARbBasketGdFlag[16], image: ImagePool.Basket Green
        p3560616238: HMI_Function.MotionX
        p2738717112: HMI_Function.MotionY
    Rectangle (268,213 32x31), "%i", text variable: DSArmBasketInfo[1].iProductRecipeNo, invisible if: NOT.ARbBasketGdFlag[16]
        p3560616238: HMI_Function.MotionX
        p2738717112: HMI_Function.MotionY
    Group (242,247 55x84)
        Image (0,0 55x84), invisible if: NOT.ARbBasketGdFlag[1], image: ImagePool.Basket Green
        Rectangle (10,42 32x31), "%i", text variable: AR2sDSCv_LdConfirmBasketInfo[1,3].iProductRecipeNo, invisible if: NOT.ARbBasketGdFlag[1]
    Group (115,248 55x84)
        Image (0,0 55x84), invisible if: NOT AR2sDSCv_LdConfirmBasketInfo[1,2].bAvailibility, image: ImagePool.Basket Green
        Rectangle (11,41 32x31), "%i", text variable: AR2sDSCv_LdConfirmBasketInfo[1,2].iProductRecipeNo, invisible if: NOT AR2sDSCv_LdConfirmBasketInfo[1,2].bAvailibility
    Group (19,248 55x84)
        Image (0,0 55x84), invisible if: NOT AR2sDSCv_LdConfirmBasketInfo[1,1].bAvailibility, image: ImagePool.Basket Green
        Rectangle (11,42 32x31), "%i", text variable: AR2sDSCv_LdConfirmBasketInfo[1,1].iProductRecipeNo, invisible if: NOT AR2sDSCv_LdConfirmBasketInfo[1,1].bAvailibility
    Group (67,193 55x84)
        Image (0,0 55x84), invisible if: NOT AR2sDSCv_LdTransferBasketInfo[1,1].bAvailibility, image: ImagePool.Basket Blue
        Rectangle (13,40 32x31), "%i", text variable: AR2sDSCv_LdTransferBasketInfo[1,1].iProductRecipeNo, invisible if: NOT AR2sDSCv_LdTransferBasketInfo[1,1].bAvailibility
    Group (163,194 55x84)
        Image (0,0 55x84), invisible if: NOT AR2sDSCv_LdTransferBasketInfo[1,2].bAvailibility, image: ImagePool.Basket Blue
        Rectangle (12,43 32x31), "%i", text variable: AR2sDSCv_LdTransferBasketInfo[1,2].iProductRecipeNo, invisible if: NOT AR2sDSCv_LdTransferBasketInfo[1,2].bAvailibility
    Group (243,266 51x51), invisible if: NOT bBlockBasketEnter
        Ellipse (0,0 51x51)
        Rectangle (3,20 45x10)
    Lamp1 (30,333 13x13), variable: ARbDI[eX13000_LoadingConveyorSensor_Feed], style: Lamp-Lamp1-Blue
    Lamp1 (155,333 13x13), variable: ARbDI[eX13001_LoadingConveyorSensor_Index], style: Lamp-Lamp1-Blue
    Lamp1 (1111,243 13x13), variable: ARbDI[eX12101_Stn06SlidingDoorRs01_Unclamp], style: Lamp-Lamp1-Blue
    Lamp1 (1111,271 13x13), variable: ARbDI[eX12100_Stn06SlidingDoorRs01_Clamp], style: Lamp-Lamp1-Blue
    Lamp1 (1269,274 13x13), variable: ARbDI[eX12102_Stn06SlidingDoorRs02_Clamp], style: Lamp-Lamp1-Blue
    Lamp1 (1269,243 13x13), variable: ARbDI[eX12103_Stn06SlidingDoorRs02_Unclamp], style: Lamp-Lamp1-Blue
    Rectangle (1124,222 150x16), invisible if: NOT ARbDI[eX12008_Stn06SlidingDoorRs_Close]
END_VISUALIZATION

// ---- VISUs/Popup_Machine_Manual.TcVIS
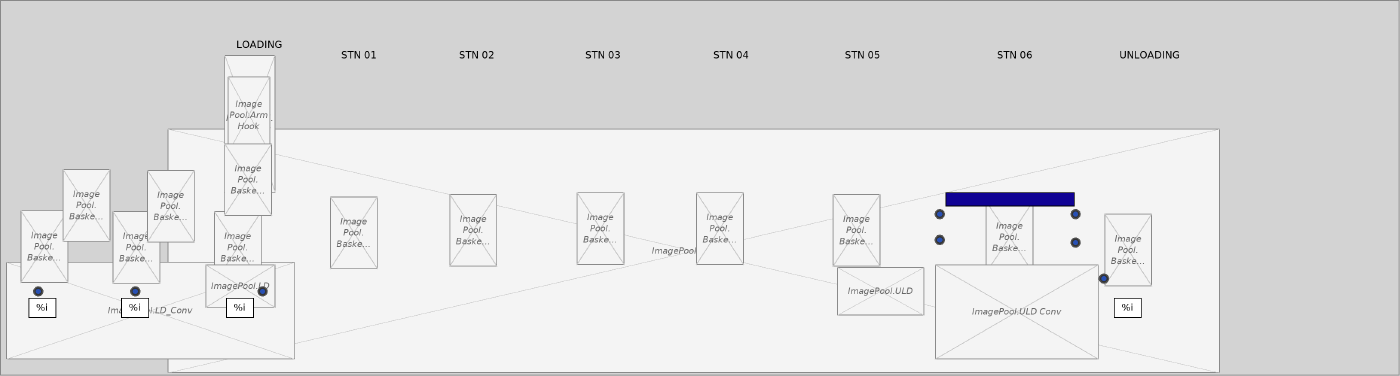
VISUALIZATION Popup_Machine_Manual  // 1629x438
    Rectangle (0,0 1629x438)
    Image (195,150 1224x284), image: ImagePool.Machine
    Label (378,44 80x40), "STN 01"
    Label (515,44 80x40), "STN 02"
    Label (662,44 80x40), "STN 03"
    Label (811,44 80x40), "STN 04"
    Label (964,44 80x40), "STN 05"
    Label (1141,44 80x40), "STN 06"
    Label (251,32 102x40), "LOADING"
    Label (1285,44 106x40), "UNLOADING"
    Group (384,229 55x84)
        Image (0,0 55x84), invisible if: NOT.ARbBasketBdFlag[2], image: ImagePool.Basket Red
            OnMouseDown: execute { DSStnBasketInfo[1].iProductRecipeNo:=0; }
        Image (0,0 55x84), invisible if: NOT.ARbBasketGdFlag[2], image: ImagePool.Basket Green
            OnMouseDown: execute { DSStnBasketInfo[1].iProductRecipeNo:=0; }
    Group (523,226 55x84)
        Image (0,0 55x84), invisible if: NOT.ARbBasketBdFlag[3], image: ImagePool.Basket Red
            OnMouseDown: execute { DSStnBasketInfo[2].iProductRecipeNo:=0; }
        Image (0,0 55x84), invisible if: NOT.ARbBasketGdFlag[3], image: ImagePool.Basket Green
            OnMouseDown: execute { DSStnBasketInfo[2].iProductRecipeNo:=0; }
    Group (671,224 55x84)
        Image (0,0 55x84), invisible if: NOT.ARbBasketBdFlag[4], image: ImagePool.Basket Red
            OnMouseDown: execute { DSStnBasketInfo[3].iProductRecipeNo:=0; }
        Image (0,0 55x84), invisible if: NOT.ARbBasketGdFlag[4], image: ImagePool.Basket Green
            OnMouseDown: execute { DSStnBasketInfo[3].iProductRecipeNo:=0; }
    Group (810,224 55x84)
        Image (0,0 55x84), invisible if: NOT.ARbBasketBdFlag[5], image: ImagePool.Basket Red
            OnMouseDown: execute { DSStnBasketInfo[4].iProductRecipeNo:=0; }
        Image (0,0 55x84), invisible if: NOT.ARbBasketGdFlag[5], image: ImagePool.Basket Green
            OnMouseDown: execute { DSStnBasketInfo[4].iProductRecipeNo:=0; }
    Group (969,226 55x84)
        Image (0,0 55x84), invisible if: NOT.ARbBasketBdFlag[6], image: ImagePool.Basket Red
            OnMouseDown: execute { DSStnBasketInfo[5].iProductRecipeNo:=0; }
        Image (0,0 55x84), invisible if: NOT.ARbBasketGdFlag[6], image: ImagePool.Basket Green
            OnMouseDown: execute { DSStnBasketInfo[5].iProductRecipeNo:=0; }
    Group (1147,234 55x84)
        Image (0,0 55x84), invisible if: NOT.ARbBasketBdFlag[7], image: ImagePool.Basket Red
            OnMouseDown: execute { DSStnBasketInfo[6].iProductRecipeNo:=0; }
        Image (0,0 55x84), invisible if: NOT.ARbBasketGdFlag[7], image: ImagePool.Basket Green
            OnMouseDown: execute { DSStnBasketInfo[6].iProductRecipeNo:=0; }
    Image (7,305 336x113), image: ImagePool.LD_Conv
    Image (249,246 55x84), invisible if: NOT.ARbBasketGdFlag[1], image: ImagePool.Basket Green
        OnMouseDown: execute { AR2sDSCv_LdConfirmBasketInfo[1,3].iProductRecipeNo:=0; }
    Image (24,245 55x84), invisible if: NOT AR2sDSCv_LdConfirmBasketInfo[1,1].bAvailibility, image: ImagePool.Basket Green
        OnMouseDown: execute { AR2sDSCv_LdConfirmBasketInfo[1,1].iProductRecipeNo:=0; }
    Image (239,308 81x50), image: ImagePool.LD
    Image (261,64 59x160), text variable: DSArmBasketInfo[1].iProductRecipeNo, image: ImagePool.Arm Body
        p3560616238: HMI_Function.MotionX
        OnMouseDown: write the text variable via VisuDialogs.Numpad
    Image (265,89 49x90), text variable: DSArmBasketInfo[1].iProductRecipeNo, image: ImagePool.Arm Hook
        p3560616238: HMI_Function.MotionX
        p2738717112: HMI_Function.MotionY
        OnMouseDown: write the text variable via VisuDialogs.Numpad
    Image (261,167 55x84), invisible if: NOT.ARbBasketBdFlag[16], image: ImagePool.Basket Red
        p3560616238: HMI_Function.MotionX
        p2738717112: HMI_Function.MotionY
        OnMouseDown: execute { DSArmBasketInfo[1].iProductRecipeNo:=0; }
    Image (261,167 55x84), invisible if: NOT.ARbBasketGdFlag[16], image: ImagePool.Basket Green
        p2738717112: HMI_Function.MotionY
        p3560616238: HMI_Function.MotionX
        OnMouseDown: execute { DSArmBasketInfo[1].iProductRecipeNo:=0; }
    Image (974,311 101x56), image: ImagePool.ULD
    Image (131,246 55x84), invisible if: NOT AR2sDSCv_LdConfirmBasketInfo[1,2].bAvailibility, image: ImagePool.Basket Green
        OnMouseDown: execute { AR2sDSCv_LdConfirmBasketInfo[1,2].iProductRecipeNo:=0; }
    Image (73,197 55x84), invisible if: NOT AR2sDSCv_LdTransferBasketInfo[1,1].bAvailibility, image: ImagePool.Basket Blue
        OnMouseDown: execute { AR2sDSCv_LdTransferBasketInfo[1,1].iProductRecipeNo:=0; }
    Image (171,198 55x84), invisible if: NOT AR2sDSCv_LdTransferBasketInfo[1,2].bAvailibility, image: ImagePool.Basket Blue
        OnMouseDown: execute { AR2sDSCv_LdTransferBasketInfo[1,2].iProductRecipeNo:=0;; }
    Image (1285,249 55x84), invisible if: NOT.ARbBasketBdFlag[12], image: ImagePool.Basket Red
        OnMouseDown: execute { AR2sDSCv_UldConfirmBasketInfo[1,1].iProductRecipeNo:=0; }
    Image (1285,249 55x84), invisible if: NOT.ARbBasketGdFlag[12], image: ImagePool.Basket Green
        OnMouseDown: execute { AR2sDSCv_UldConfirmBasketInfo[1,1].iProductRecipeNo:=0; }
    Image (1088,308 190x110), image: ImagePool.ULD Conv
    Lamp1 (1278,318 13x13), variable: ARbDI[eX12011_UnloadingSensor_BasketDetection], style: Lamp-Lamp1-Blue
    Rectangle (1296,347 32x23), "%i", text variable: AR2sDSCv_UldConfirmBasketInfo[1,1].iProductRecipeNo
        OnMouseDown: write the text variable via VisuDialogs.Numpad
    Rectangle (263,347 32x23), "%i", text variable: AR2sDSCv_LdConfirmBasketInfo[1,3].iProductRecipeNo
        OnMouseDown: write the text variable via VisuDialogs.Numpad
    Rectangle (141,347 32x23), "%i", text variable: AR2sDSCv_LdConfirmBasketInfo[1,2].iProductRecipeNo
        OnMouseDown: write the text variable via VisuDialogs.Numpad
    Rectangle (33,347 32x23), "%i", text variable: AR2sDSCv_LdConfirmBasketInfo[1,1].iProductRecipeNo
        OnMouseDown: write the text variable via VisuDialogs.Numpad
    Lamp1 (299,333 13x13), variable: ARbDI[eX13002_LoadingConveyorSensor_Pick], style: Lamp-Lamp1-Blue
    Lamp1 (38,333 13x13), variable: ARbDI[eX13000_LoadingConveyorSensor_Feed], style: Lamp-Lamp1-Blue
    Lamp1 (151,333 13x13), variable: ARbDI[eX13001_LoadingConveyorSensor_Index], style: Lamp-Lamp1-Blue
    Lamp1 (1087,243 13x13), variable: ARbDI[eX12101_Stn06SlidingDoorRs01_Unclamp], style: Lamp-Lamp1-Blue
    Lamp1 (1087,273 13x13), variable: ARbDI[eX12100_Stn06SlidingDoorRs01_Clamp], style: Lamp-Lamp1-Blue
    Lamp1 (1245,276 13x13), variable: ARbDI[eX12102_Stn06SlidingDoorRs02_Clamp], style: Lamp-Lamp1-Blue
    Lamp1 (1245,243 13x13), variable: ARbDI[eX12103_Stn06SlidingDoorRs02_Unclamp], style: Lamp-Lamp1-Blue
    Rectangle (1100,224 150x16), invisible if: NOT ARbDI[eX12008_Stn06SlidingDoorRs_Close]
END_VISUALIZATION

// ---- VISUs/Popup_MenuPage.TcVIS
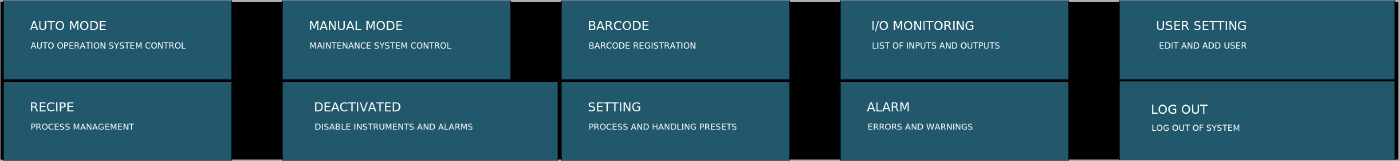
VISUALIZATION Popup_MenuPage  // 1922x222
    Rectangle (-2,2 1922x218)
    Rectangle (3,2 1x218)
        p3528305787: HMI_Ctrl.ANIMATION
    Group (1153,112 379x110)
        OnMouseClick: execute { iBufferPage := 8; }
        Rectangle (0,0 314x110)
            OnMouseClick: change screen: Alarm_Page
        Label (34,9 221x53), "ALARM"
        Label (35,32 190x62), "ERRORS AND WARNINGS"
    Group (1153,0 379x110)
        OnMouseClick: execute { iBufferPage := 4; }
        Rectangle (0,0 314x110)
            OnMouseClick: change screen: IO_Monitoring
        Label (40,9 221x53), "I/O MONITORING"
        Label (41,32 249x62), "LIST OF INPUTS AND OUTPUTS"
    Group (1536,111 379x110)
        OnMouseClick: execute { iBufferPage:=10; }
        Rectangle (0,0 379x110)
            OnMouseDown: execute { iBufferPage:=10; }
        Label (41,27 267x26), "LOG OUT"
        Label (42,50 229x31), "LOG OUT OF SYSTEM"
    Group (4,0 379x110)
        OnMouseClick: execute { iBufferPage := 1; }
        Rectangle (0,0 314x110)
        Label (34,9 221x53), "AUTO MODE"
        Label (35,32 279x62), "AUTO OPERATION SYSTEM CONTROL"
    Group (4,112 379x110), input disabled if: iCurrentUserGroupID<3
        OnMouseClick: execute { iBufferPage := 5; }
        Rectangle (0,0 314x110)
        Label (34,9 221x53), "RECIPE"
        Label (35,32 279x62), "PROCESS MANAGEMENT"
    Group (387,0 379x110), input disabled if: iCurrentUserGroupID<2 OR bMainOnOff
        OnMouseClick: execute { iBufferPage := 2; }
        Rectangle (0,0 314x110)
        Label (34,9 221x53), "MANUAL MODE"
        Label (35,32 279x62), "MAINTENANCE SYSTEM CONTROL"
    Group (387,112 379x110), input disabled if: iCurrentUserGroupID<2
        OnMouseClick: execute { iBufferPage := 6; }
        Rectangle (0,0 379x110)
        Label (41,9 267x53), "DEACTIVATED"
        Label (42,32 337x62), "DISABLE INSTRUMENTS AND ALARMS"
    Group (770,0 379x110), input disabled if: iCurrentUserGroupID<3
        OnMouseClick: execute { iBufferPage := 3; }
        Rectangle (0,0 314x110)
            OnMouseClick: change screen: Barcode_Page
        Label (34,9 221x53), "BARCODE"
        Label (35,32 279x62), "BARCODE REGISTRATION"
    Group (770,112 379x110), input disabled if: iCurrentUserGroupID<3
        OnMouseClick: execute { iBufferPage := 7; }
        Rectangle (0,0 314x110)
        Label (34,9 221x53), "SETTING"
        Label (35,32 279x62), "PROCESS AND HANDLING PRESETS"
    Group (1536,0 379x110), input disabled if: iCurrentUserGroupID<4
        OnMouseClick: execute { iBufferPage:=11; }
        Rectangle (0,0 379x110)
            OnMouseClick: change screen: IO_Monitoring
        Label (48,9 267x53), "USER SETTING"
        Label (52,32 301x62), "EDIT AND ADD USER"
END_VISUALIZATION

// ---- VISUs/RecipeNo.TcTLO
TEXTLIST RecipeNo
  1 = '1'
  2 = '2'
  3 = '3'
  4 = '4'
  5 = '5'
  6 = '6'
  7 = '7'
  8 = '8'
  9 = '9'
  10 = '10'
  11 = '11'
  12 = '12'
  13 = '13'
  14 = '14'
  15 = '15'
  16 = '16'
  17 = '17'
  18 = '18'
  19 = '19'
  20 = '20'
   = ''
END_TEXTLIST

// ---- VISUs/RECIPE/RecipeConfiguration_Page.TcVIS
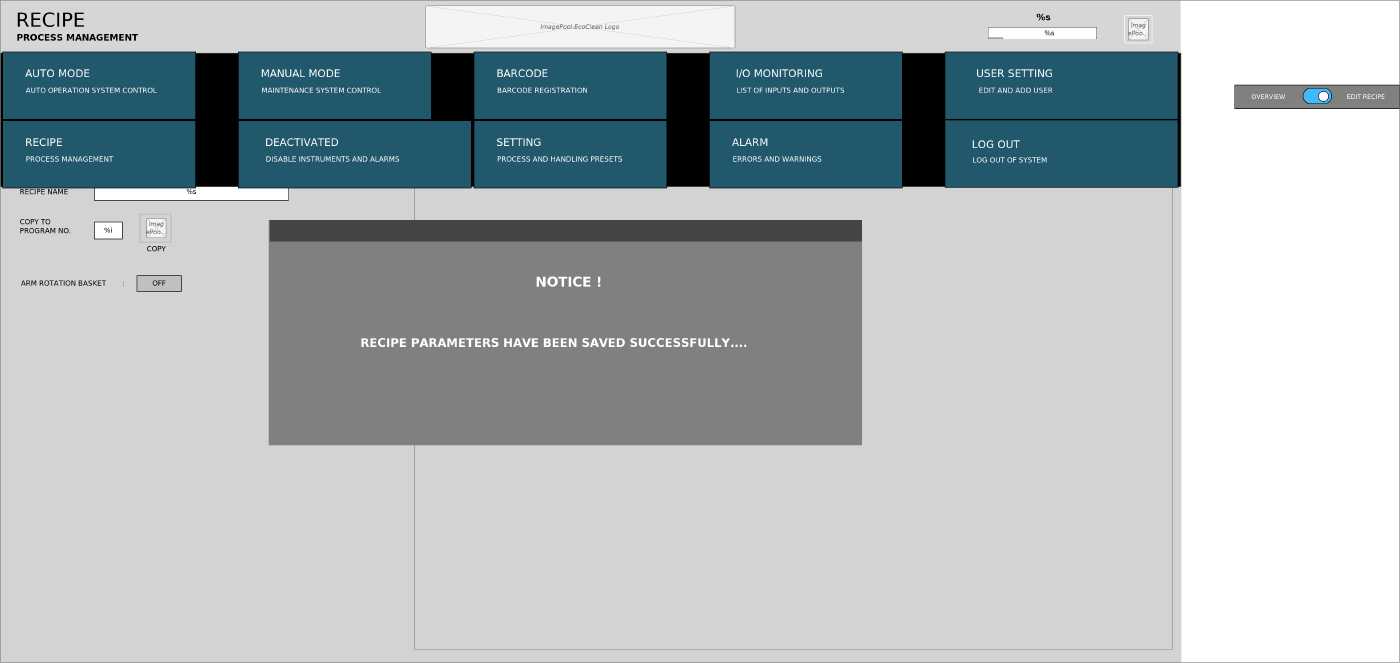
VISUALIZATION RecipeConfiguration_Page  // 2276x1079
    RoundedRectangle (245,275 1437x791)
    Rectangle (0,98 1920x981), "%i", text variable: Global_Variables_Arm_Persistent.DSA1fbPnpSequenceMemoryStore.iProductRecipeNo
    Rectangle (0,63 1920x26)
        p3528305787: HMI_Ctrl.ANIMATION3
    Rectangle (0,0 1919x85)
    Group (23,6 321x67)
        Label (0,0 267x53), "RECIPE"
        Label (1,43 320x24), "PROCESS MANAGEMENT"
    Frame (673,269 1233x788)
        shows Popup_RecipeConfiguration()
    Rectangle (799,197 136x63), "STATION"
    Rectangle (938,197 136x63), "SSER NO."
    Rectangle (1077,197 441x63), "DESCRIPTION"
    Group (1521,197 309x63)
        Rectangle (0,33 153x30), "PICK UP"
        Rectangle (156,33 153x30), "DOWN TRANSFER"
        Rectangle (0,0 309x30), "ARM PATTERN"
    Group (1828,25 45x45)
        OnMouseClick: toggle HMI_Ctrl.MenuButton
        RoundedRectangle (0,0 45x45), colour toggle: HMI_Ctrl.MenuButton
        Image (6,5 33x35), image: ImagePool.Menu Button
    Group (2007,137 269x41)
        RoundedRectangle (0,1 269x39)
        Label (1,0 108x41), "OVERVIEW"
        Label (161,0 105x41), "EDIT RECIPE"
        Group (111,6 47x26)
            OnMouseClick: change screen: Recipe_Page
            Group (0,0 47x26)
                Ellipse (0,0 26x26)
                Ellipse (21,0 26x26)
                RoundedRectangle (8,0 29x26)
            Ellipse (1,1 24x24)
            Ellipse (23,1 23x24)
            RoundedRectangle (9,1 28x24)
            Ellipse (25,5 17x17)
    Ellipse (867,123 25x25)
    Ellipse (948,123 25x25)
    Ellipse (904,130 10x10)
    Ellipse (926,130 10x10)
    Ellipse (985,130 10x10)
    Ellipse (1007,130 10x10)
    Ellipse (1029,123 25x25)
    Label (847,153 64x24), "SSUR"
    Label (928,153 64x24), "SSER"
    Label (1009,153 64x24), "CONFIG"
    Image (790,113 45x45), image: ImagePool.Previous Button
        OnMouseClick: change screen: RecipeSSER_Page
    Rectangle (26,197 403x30), "PRODUCT RECIPE CONFIGURATION"
    Label (29,253 93x24), "RECIPE NO."
    RoundedRectangle (153,251 51x28), "%i", text variable: Global_Variables_Arm_Persistent.DSA1fbPnpSequenceMemoryStore.iProductRecipeNo
        OnMouseDown: write the text variable via Default, min 1, max 40
    Label (29,300 101x24), "RECIPE NAME"
    RoundedRectangle (153,298 316x28), "%s", text variable: Global_Variables_Arm_Persistent.DSA1fbPnpSequenceMemoryStore.DsA1inPnpSequenceMemory.sDescription
        OnMouseDown: write the text variable via VisuDialogs.Keypad
    Label (29,348 110x41), "COPY TO PROGRAM NO."
    RoundedRectangle (153,361 46x28), "%i", text variable: DSA1fbPnpSequenceMemoryStore.iCopyToProductRecipeNo
        OnMouseDown: write the text variable via VisuDialogs.Numpad, min 1, max 40
    Image (691,9 504x69), image: ImagePool.EcoClean Logo
    Group (227,348 51x69), invisible if: bMainOnOff
        Label (6,45 42x24), "COPY"
        RoundedRectangle (0,0 51x46), colour toggle: DSA1fbPnpSequenceMemoryStore.bCopyPB
            tap DSA1fbPnpSequenceMemoryStore.bCopyPB
        Image (11,7 32x32), image: ImagePool.Copy Button
            OnMouseDown: execute { DSA1fbPnpSequenceMemoryStore.bCopyPB:=1; }
            OnMouseUp: execute { DSA1fbPnpSequenceMemoryStore.bCopyPB:=0; }
    Group (1606,17 179x46)
        Button (0,27 177x19), image: VisuSymbols.Symbols.AddUser
        Rectangle (25,28 150x18), "%s", text variable: fbHmiTF1800_UserlevelManagement.dsHmiUserStatus_Active.sLoginName
        Rectangle (2,0 177x22), "%s", text variable: DSLocalSystemTimeML.sCurrentDT24Hr_General
    Group (487,216 56x80), invisible if: bMainOnOff
        Label (5,52 51x28), "SAVE", invisible if: bMainOnOff
        RoundedRectangle (0,0 55x56), colour toggle: bRecipeSavePb
            tap bRecipeSavePb
        Image (11,5 34x45), image: ImagePool.Save Button
            OnMouseDown: execute { bRecipeSavePb:=1; }
            OnMouseUp: execute { bRecipeSavePb:=0; }
    Frame (437,358 964x366), invisible if: NOT stWritePersistentData.SaveHR
        shows Popup_Parameter_Saved()
    Label (31,449 183x24), "ARM ROTATION BASKET"
    Label (196,449 19x24), ":"
    Rectangle (222,448 73x26), "ON", invisible if: NOT DSA1fbPnpSequenceMemoryStore.DsA1inPnpSequenceMemory.bArmRotaryBarrelEnable
        OnMouseDown: execute { DSA1fbPnpSequenceMemoryStore.DsA1inPnpSequenceMemory.bArmRotaryBarrelEnable:=FALSE; }
    Rectangle (222,448 73x26), "OFF", invisible if: DSA1fbPnpSequenceMemoryStore.DsA1inPnpSequenceMemory.bArmRotaryBarrelEnable
        OnMouseDown: execute { DSA1fbPnpSequenceMemoryStore.DsA1inPnpSequenceMemory.bArmRotaryBarrelEnable:=TRUE; }
    Label (560,271 50x24), "CLEAR"
    RoundedRectangle (556,216 55x56), colour toggle: bProductRecipeClearPb
        tap bProductRecipeClearPb
    Image (567,222 34x40), image: ImagePool.Clear Button
        OnMouseDown: execute { bProductRecipeClearPb:=1; }
        OnMouseUp: execute { bProductRecipeClearPb:=0; }
    Frame (0,84 1918x221), invisible if: HMI_Ctrl.CloseMenuButton
        shows Popup_MenuPage()
END_VISUALIZATION

// ---- VISUs/RECIPE/RecipeSSER_Page.TcVIS
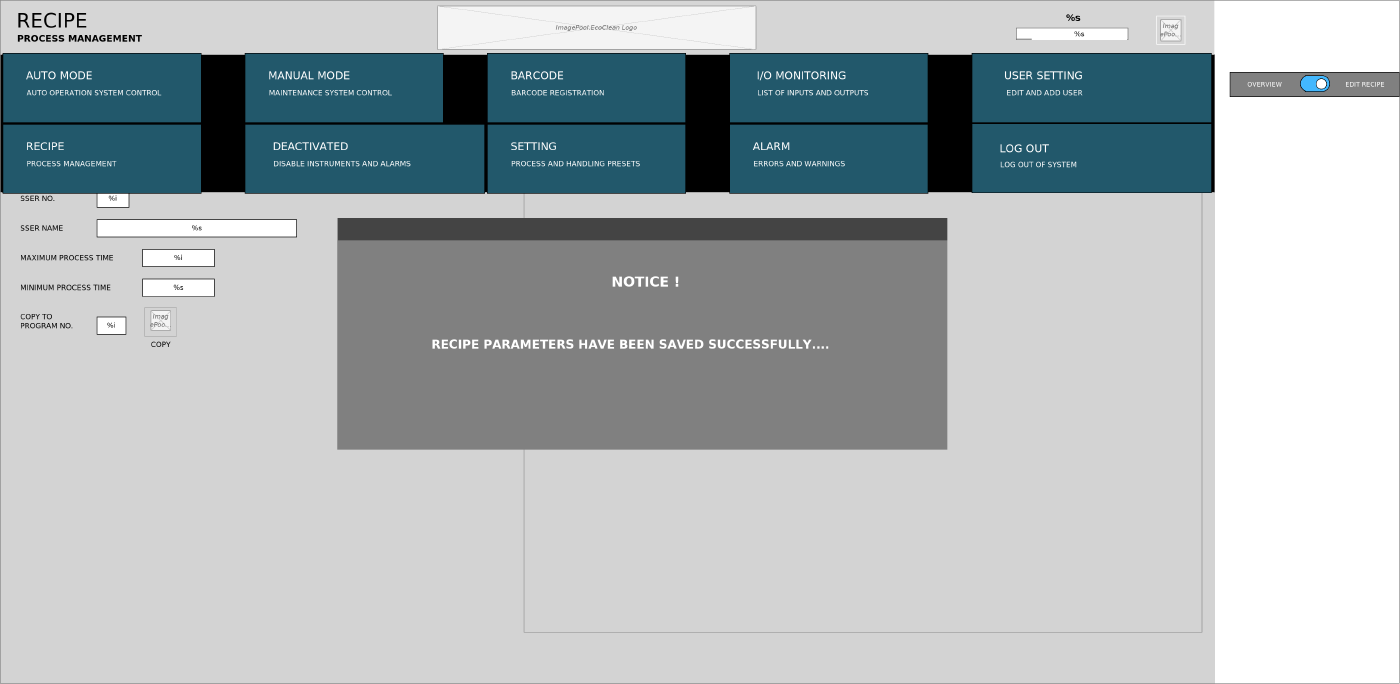
VISUALIZATION RecipeSSER_Page  // 2213x1082
    Rectangle (0,101 1920x981)
    Rectangle (0,63 1920x26)
        p3528305787: HMI_Ctrl.ANIMATION3
    Rectangle (0,0 1919x85)
    Group (23,6 321x67)
        Label (0,0 267x53), "RECIPE"
        Label (1,43 320x24), "PROCESS MANAGEMENT"
    Frame (828,265 1072x735)
        shows Popup_RecipeSSER()
    Rectangle (946,196 142x63), "SSUR NO."
    Rectangle (1092,196 445x63), "DESCRIPTION"
    Group (1828,25 45x45)
        OnMouseClick: toggle HMI_Ctrl.MenuButton
        RoundedRectangle (0,0 45x45), colour toggle: HMI_Ctrl.MenuButton
        Image (6,5 33x35), image: ImagePool.Menu Button
    Group (1944,113 269x41)
        RoundedRectangle (0,1 269x39)
        Label (1,0 108x41), "OVERVIEW"
        Label (161,0 105x41), "EDIT RECIPE"
        Group (111,6 47x26)
            OnMouseClick: change screen: Recipe_Page
            Group (0,0 47x26)
                Ellipse (0,0 26x26)
                Ellipse (21,0 26x26)
                RoundedRectangle (8,0 29x26)
            Ellipse (1,1 24x24)
            Ellipse (23,1 23x24)
            RoundedRectangle (9,1 28x24)
            Ellipse (25,5 17x17)
    Group (790,113 341x64)
        Ellipse (77,10 25x25)
        Ellipse (158,10 25x25)
        Ellipse (114,17 10x10)
        Ellipse (136,17 10x10)
        Ellipse (195,17 10x10)
        Ellipse (217,17 10x10)
        Ellipse (239,10 25x25)
        Label (57,40 64x24), "SSUR"
        Label (138,40 64x24), "SSER"
        Label (219,40 64x24), "CONFIG"
        Image (296,0 45x45), image: ImagePool.Next Button
            OnMouseClick: change screen: RecipeConfiguration_Page
        Image (0,0 45x45), image: ImagePool.Previous Button
            OnMouseClick: change screen: RecipeSSUR_Page
    Rectangle (26,197 403x30), "SEQUENCE RECIPE CONFIGURATION (SSER)"
    RoundedRectangle (26,236 292x48)
    Label (46,248 79x24), "STATION"
    ComboBoxInteger (129,245 162x30), variable: iStationNo, text list: 'TextList_Recipe'
    Label (29,302 93x24), "SSER NO."
    RoundedRectangle (153,300 51x28), "%i", text variable: DSScrMapSSER.iStationSequenceRecipeNo
        OnMouseDown: write the text variable via VisuDialogs.Numpad, min 1, max 20
    Label (29,396 174x24), "MAXIMUM PROCESS TIME"
    RoundedRectangle (225,394 114x28), "%i", text variable: DSScrMapSSER.DsStationSequenceRecipeMemory.iProcessMaxTime
        OnMouseDown: write the text variable via VisuDialogs.Numpad, min 1, max 9999
    Label (29,443 174x24), "MINIMUM PROCESS TIME"
    RoundedRectangle (225,441 114x28), "%s", text variable: DSScrMapSSER.DsStationSequenceRecipeMemory.iProcessMinTime
        OnMouseDown: write the text variable via VisuDialogs.Numpad, min 1, max 9999
    Label (29,349 101x24), "SSER NAME"
    RoundedRectangle (153,347 316x28), "%s", text variable: DSScrMapSSER.sStationSequenceRecipeDescription
        OnMouseDown: write the text variable via VisuDialogs.Keypad
    Label (29,488 110x41), "COPY TO PROGRAM NO."
    RoundedRectangle (153,501 46x28), "%i", text variable: DSScrMapSSER.iCopyToSubRecipeNo
        OnMouseDown: write the text variable via VisuDialogs.Numpad, min 1, max 20
    Rectangle (830,196 113x63), "STEP"
    Image (691,9 504x69), image: ImagePool.EcoClean Logo
    Rectangle (1540,196 153x63), "CYCLE"
    Rectangle (1696,196 175x63), "REPEAT FROM STEP NO."
    Group (228,486 51x71), invisible if: bMainOnOff
        Label (5,47 42x24), "COPY"
        RoundedRectangle (0,0 51x46), colour toggle: DSScrMapSSER.bCopyPB
            tap DSScrMapSSER.bCopyPB
        Image (10,5 32x32), image: ImagePool.Copy Button
            OnMouseDown: execute { DSScrMapSSER.bCopyPB:=1; }
            OnMouseUp: execute { DSScrMapSSER.bCopyPB:=0; }
    Group (1606,17 179x46)
        Button (0,27 177x19), image: VisuSymbols.Symbols.AddUser
        Rectangle (25,28 150x18), "%s", text variable: fbHmiTF1800_UserlevelManagement.dsHmiUserStatus_Active.sLoginName
        Rectangle (2,0 177x22), "%s", text variable: DSLocalSystemTimeML.sCurrentDT24Hr_General
    Group (517,196 56x80), invisible if: bMainOnOff
        Label (5,52 51x28), "SAVE", invisible if: bMainOnOff
        RoundedRectangle (0,0 55x56), colour toggle: bRecipeSavePb
            tap bRecipeSavePb
        Image (11,5 34x45), image: ImagePool.Save Button
            OnMouseDown: execute { bRecipeSavePb:=1; }
            OnMouseUp: execute { bRecipeSavePb:=0; }
    Frame (533,345 964x366), invisible if: NOT stWritePersistentData.SaveHR
        shows Popup_Parameter_Saved()
    Label (585,250 60x24), "CLEAR"
    RoundedRectangle (589,197 51x53), colour toggle: bRecipeClearInd_SSER
        tap bBufferClearPB_SSER[iStationNo]
    Image (596,203 34x40), image: ImagePool.Clear Button
        OnMouseDown: execute { bBufferClearPB_SSER[iStationNo]:=1; }
        OnMouseUp: execute { bBufferClearPB_SSER[iStationNo]:=0; }
    Frame (0,84 1918x221), invisible if: HMI_Ctrl.CloseMenuButton
        shows Popup_MenuPage()
END_VISUALIZATION

// ---- VISUs/RECIPE/RecipeSSUR_Page.TcVIS
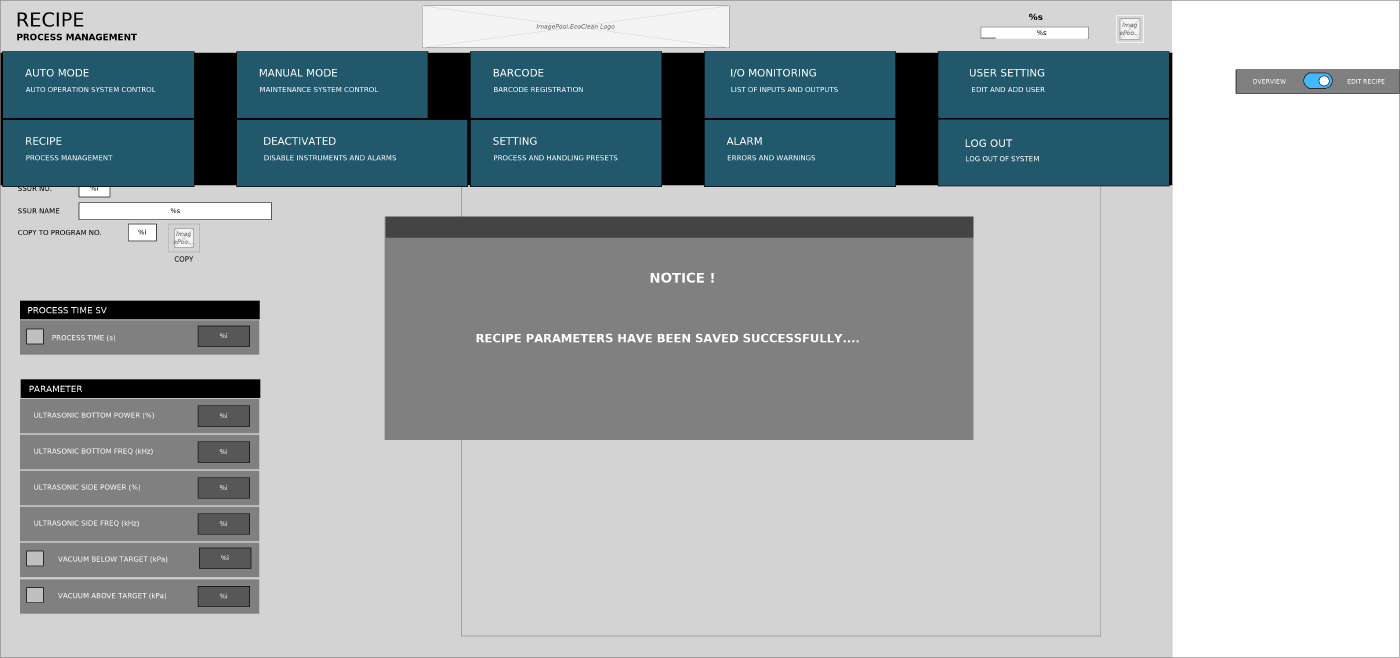
VISUALIZATION RecipeSSUR_Page  // 2293x1079
    Rectangle (0,98 1920x981)
    Rectangle (0,63 1920x26)
        p3528305787: HMI_Ctrl.ANIMATION3
    Rectangle (0,0 1919x85)
    Group (23,6 321x67)
        Label (0,0 267x53), "RECIPE"
        Label (1,43 320x24), "PROCESS MANAGEMENT"
    Frame (755,198 1048x845)
        shows Recipe_AllStation_SSUR()
    RoundedRectangle (25,235 292x48)
    Label (45,247 79x24), "STATION"
    Label (26,297 101x24), "SSUR NO."
    RoundedRectangle (129,295 51x28), "%i", text variable: DSScrMapSSUR.iSubRecipeNo
        OnMouseDown: write the text variable via VisuDialogs.Numpad, min 1, max 20
    Label (26,334 101x24), "SSUR NAME"
    RoundedRectangle (129,332 316x28), "%s", text variable: DSScrMapSSUR.sSubRecipeDescription
        OnMouseDown: write the text variable via VisuDialogs.Keypad
    Rectangle (24,197 433x30), "SUB PROCESS RECIPE CONFIGURATION (SSUR)"
    Label (26,361 156x41), "COPY TO PROGRAM NO."
    RoundedRectangle (210,367 46x28), "%i", text variable: DSScrMapSSUR.iCopyToSubRecipeNo
        OnMouseDown: write the text variable via VisuDialogs.Numpad, min 1, max 20
    ComboBoxInteger (128,244 162x30), variable: iStationNo, text list: 'TextList_Recipe'
    Group (1828,25 45x45)
        OnMouseClick: toggle HMI_Ctrl.MenuButton
        RoundedRectangle (0,0 45x45), colour toggle: HMI_Ctrl.MenuButton
        Image (6,5 33x35), image: ImagePool.Menu Button
    Group (2024,113 269x41)
        RoundedRectangle (0,1 269x39)
        Label (1,0 108x41), "OVERVIEW"
        Label (161,0 105x41), "EDIT RECIPE"
        Group (111,6 47x26)
            OnMouseClick: change screen: Recipe_Page
            Group (0,0 47x26)
                Ellipse (0,0 26x26)
                Ellipse (21,0 26x26)
                RoundedRectangle (8,0 29x26)
            Ellipse (1,1 24x24)
            Ellipse (23,1 23x24)
            RoundedRectangle (9,1 28x24)
            Ellipse (25,5 17x17)
    Ellipse (867,123 25x25)
    Ellipse (948,123 25x25)
    Ellipse (904,130 10x10)
    Ellipse (926,130 10x10)
    Ellipse (985,130 10x10)
    Ellipse (1007,130 10x10)
    Ellipse (1029,123 25x25)
    Label (847,153 64x24), "SSUR"
    Label (928,153 64x24), "SSER"
    Label (1009,153 64x24), "CONFIG"
    Image (1086,113 45x45), image: ImagePool.Next Button
        OnMouseClick: change screen: RecipeSSER_Page
    Rectangle (33,525 391x56)
    Label (82,546 150x16), "PROCESS TIME (s)"
    Rectangle (324,534 85x34), "%i", text variable: DSScrMapSSUR.DsSubRecipeMemory.iComCon5ProcessTimer, invisible if: NOT.DSScrMapSSUR.DsSubRecipeMemory.bComCon20EnProcessTimer
        OnMouseDown: write the text variable via VisuDialogs.Numpad, min 0, max 9999
    Rectangle (33,493 392x30)
    Label (42,501 304x16), "PROCESS TIME SV"
    Rectangle (43,539 28x25)
        toggle DSScrMapSSUR.DsSubRecipeMemory.bComCon20EnProcessTimer
    Label (46,719 150x16)
    Label (46,687 150x16)
    Rectangle (33,654 391x56), invisible if: NOT DSScrMapSSUR.DsSubRecipeMemory.bOut3EnProTankBottomUltrasonicA
    Label (52,673 240x16), "ULTRASONIC BOTTOM POWER (%)", invisible if: NOT DSScrMapSSUR.DsSubRecipeMemory.bOut3EnProTankBottomUltrasonicA
    Rectangle (324,665 85x34), "%i", text variable: DSScrMapSSUR.DsSubRecipeMemory.iOut3ProTankBtmUsAPwrPercent, invisible if: NOT DSScrMapSSUR.DsSubRecipeMemory.bOut3EnProTankBottomUltrasonicA
        OnMouseDown: write the text variable via VisuDialogs.Numpad, min 10, max 100
    Rectangle (33,713 391x56), invisible if: NOT DSScrMapSSUR.DsSubRecipeMemory.bOut3EnProTankBottomUltrasonicA
    Label (52,732 239x16), "ULTRASONIC BOTTOM FREQ (kHz)", invisible if: NOT DSScrMapSSUR.DsSubRecipeMemory.bOut3EnProTankBottomUltrasonicA
    Rectangle (324,724 85x34), "%i", text variable: .DSScrMapSSUR.DsSubRecipeMemory.iOut8ProTankBtmUsAkHz, invisible if: NOT DSScrMapSSUR.DsSubRecipeMemory.bOut3EnProTankBottomUltrasonicA
        tap bFreqBtmChange[iStationNo]
    Rectangle (34,622 392x30)
    Label (44,630 304x16), "PARAMETER"
    Image (691,9 504x69), image: ImagePool.EcoClean Logo
    Group (276,367 51x70), invisible if: bMainOnOff
        RoundedRectangle (0,0 51x46), colour toggle: DSScrMapSSUR.bCopyPB
            tap DSScrMapSSUR.bCopyPB
        Image (9,7 32x32), image: ImagePool.Copy Button
            OnMouseDown: execute { DSScrMapSSUR.bCopyPB:=1; }
            OnMouseUp: execute { DSScrMapSSUR.bCopyPB:=0; }
        Label (4,46 42x24), "COPY"
    Group (1606,17 179x46)
        Button (0,27 177x19), image: VisuSymbols.Symbols.AddUser
        Rectangle (25,28 150x18), "%s", text variable: fbHmiTF1800_UserlevelManagement.dsHmiUserStatus_Active.sLoginName
        Rectangle (2,0 177x22), "%s", text variable: DSLocalSystemTimeML.sCurrentDT24Hr_General
    Group (527,196 56x80), invisible if: bMainOnOff
        Label (5,52 51x28), "SAVE", invisible if: bMainOnOff
        RoundedRectangle (0,0 55x56), colour toggle: bRecipeSavePb
            tap bRecipeSavePb
        Image (11,5 34x45), image: ImagePool.Save Button
            OnMouseDown: execute { bRecipeSavePb:=1; }
            OnMouseUp: execute { bRecipeSavePb:=0; }
    Frame (630,355 964x366), invisible if: NOT stWritePersistentData.SaveHR
        shows Popup_Parameter_Saved()
    Rectangle (33,890 391x56), invisible if: iStationNo<>6 OR NOT DSScrMapSSUR.DsSubRecipeMemory.bOut11EnVacuumPump
    Label (92,909 221x16), "VACUUM BELOW TARGET (kPa)", invisible if: iStationNo<>6 OR NOT DSScrMapSSUR.DsSubRecipeMemory.bOut11EnVacuumPump
    Rectangle (326,898 85x34), "%i", text variable: DSScrMapSSUR.DsSubRecipeMemory.iComCon1TargetVacuumLevel, invisible if: NOT DSScrMapSSUR.DsSubRecipeMemory.bComCon11EnBelowTargetVacuumLevel
        OnMouseDown: write the text variable via VisuDialogs.Numpad, min -120, max 10
    Rectangle (33,950 391x56), invisible if: iStationNo<>6 OR NOT DSScrMapSSUR.DsSubRecipeMemory.bOut11EnVacuumPump
    Label (92,969 214x16), "VACUUM ABOVE TARGET (kPa)", invisible if: iStationNo<>6 OR NOT DSScrMapSSUR.DsSubRecipeMemory.bOut11EnVacuumPump
    Rectangle (324,961 85x34), "%i", text variable: DSScrMapSSUR.DsSubRecipeMemory.iComCon1TargetVacuumLevel, invisible if: NOT DSScrMapSSUR.DsSubRecipeMemory.bComCon12EnAboveTargetVacuumLevel
        OnMouseDown: write the text variable via VisuDialogs.Numpad, min -120, max 10
    Label (46,837 150x16)
    Label (46,805 150x16)
    Rectangle (33,772 391x56), invisible if: NOT DSScrMapSSUR.DsSubRecipeMemory.bOut6EnProTankSideUltrasonicA
    Label (52,791 212x16), "ULTRASONIC SIDE POWER (%)", invisible if: NOT DSScrMapSSUR.DsSubRecipeMemory.bOut6EnProTankSideUltrasonicA
    Rectangle (324,783 85x34), "%i", text variable: DSScrMapSSUR.DsSubRecipeMemory.iOut6ProTankSideUsAPwrPercent, invisible if: NOT DSScrMapSSUR.DsSubRecipeMemory.bOut6EnProTankSideUltrasonicA
        OnMouseDown: write the text variable via VisuDialogs.Numpad, min 10, max 100
    Rectangle (33,831 391x56), invisible if: NOT DSScrMapSSUR.DsSubRecipeMemory.bOut6EnProTankSideUltrasonicA
    Label (52,850 217x16), "ULTRASONIC SIDE FREQ (kHz)", invisible if: NOT DSScrMapSSUR.DsSubRecipeMemory.bOut6EnProTankSideUltrasonicA
    Rectangle (324,842 85x34), "%i", text variable: .DSScrMapSSUR.DsSubRecipeMemory.iOut11ProTankSideUsAkHz, invisible if: NOT DSScrMapSSUR.DsSubRecipeMemory.bOut6EnProTankSideUltrasonicA
        tap bFreqSideChange[iStationNo]
    Rectangle (43,903 28x25), invisible if: iStationNo<>6 OR NOT DSScrMapSSUR.DsSubRecipeMemory.bOut11EnVacuumPump
        toggle DSScrMapSSUR.DsSubRecipeMemory.bComCon11EnBelowTargetVacuumLevel
    Rectangle (43,963 28x25), invisible if: iStationNo<>6 OR NOT DSScrMapSSUR.DsSubRecipeMemory.bOut11EnVacuumPump
        toggle DSScrMapSSUR.DsSubRecipeMemory.bComCon12EnAboveTargetVacuumLevel
    RoundedRectangle (595,198 51x53), colour toggle: bRecipeClearInd_SSER
        tap bBufferClearPB_SSUR[iStationNo]
    Label (597,251 50x24), "CLEAR"
    Image (605,204 34x40), image: ImagePool.Clear Button
        OnMouseDown: execute { bBufferClearPB_SSUR[iStationNo]:=1; }
        OnMouseUp: execute { bBufferClearPB_SSUR[iStationNo]:=0; }
    Frame (0,84 1918x221), invisible if: HMI_Ctrl.CloseMenuButton
        shows Popup_MenuPage()
END_VISUALIZATION

// ---- VISUs/RECIPE/Recipe_Page.TcVIS
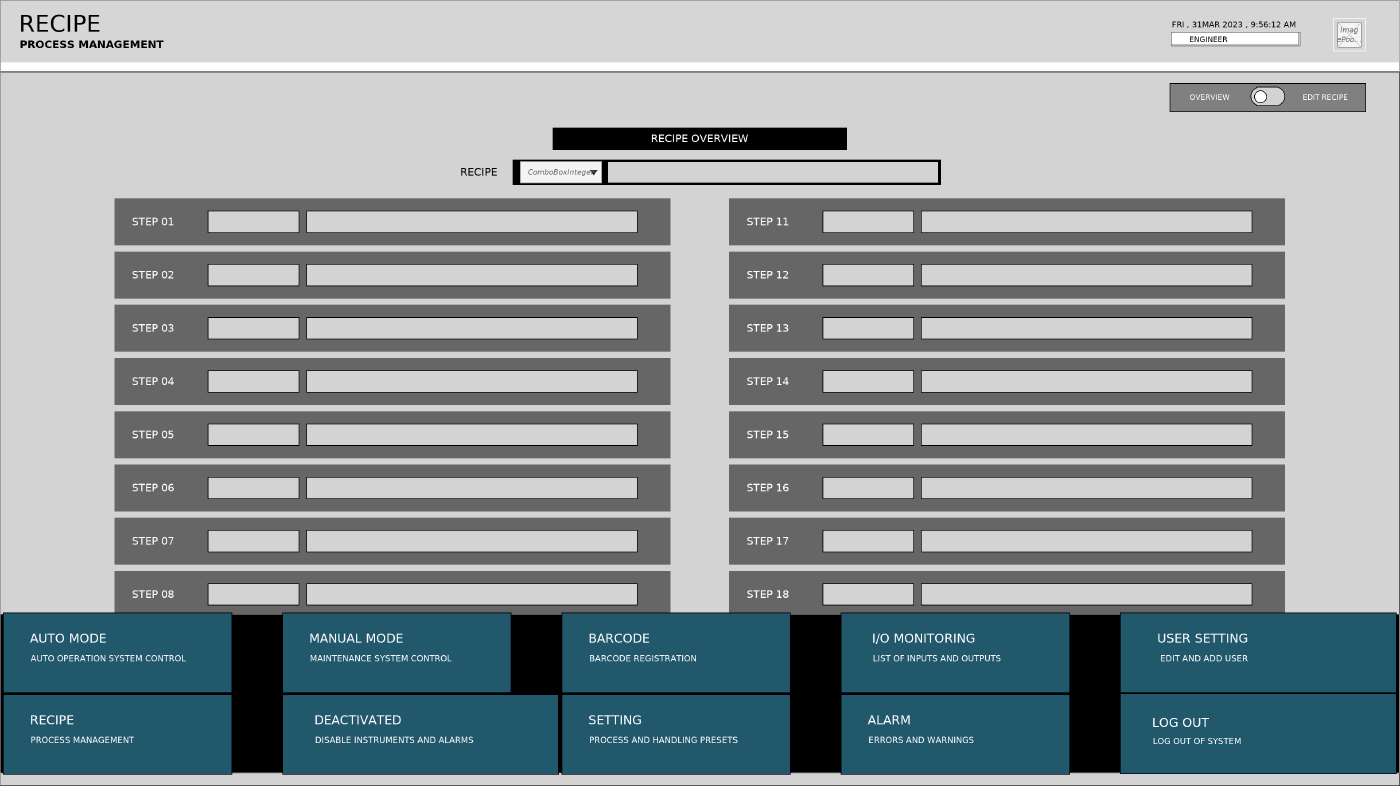
VISUALIZATION Recipe_Page  // 1920x1078
    Rectangle (0,98 1920x980)
    Rectangle (0,63 1920x26)
        p3528305787: HMI_Ctrl.ANIMATION3
    Rectangle (0,0 1919x85)
    Label (23,6 267x53), "RECIPE"
    Label (24,49 320x24), "PROCESS MANAGEMENT"
    Group (1604,25 188x38)
        Label (0,0 188x18), "FRI , 31MAR 2023 , 9:56:12 AM"
        Button (2,19 177x19), image: VisuSymbols.Symbols.AddUser
        Label (24,23 91x12), "ENGINEER"
    RoundedRectangle (157,272 762x64)
    Label (178,292 103x24), "STEP 01"
    RoundedRectangle (285,289 125x30)
    RoundedRectangle (420,289 454x30)
    RoundedRectangle (157,345 762x64)
    Label (178,365 103x24), "STEP 02"
    RoundedRectangle (285,362 125x30)
    RoundedRectangle (420,362 454x30)
    RoundedRectangle (157,418 762x64)
    Label (178,438 103x24), "STEP 03"
    RoundedRectangle (285,435 125x30)
    RoundedRectangle (420,435 454x30)
    RoundedRectangle (157,491 762x64)
    Label (178,511 103x24), "STEP 04"
    RoundedRectangle (285,508 125x30)
    RoundedRectangle (420,508 454x30)
    RoundedRectangle (157,564 762x64)
    Label (178,584 103x24), "STEP 05"
    RoundedRectangle (285,581 125x30)
    RoundedRectangle (420,581 454x30)
    RoundedRectangle (157,637 762x64)
    Label (178,657 103x24), "STEP 06"
    RoundedRectangle (285,654 125x30)
    RoundedRectangle (420,654 454x30)
    RoundedRectangle (157,710 762x64)
    Label (178,730 103x24), "STEP 07"
    RoundedRectangle (285,727 125x30)
    RoundedRectangle (420,727 454x30)
    RoundedRectangle (157,783 762x64)
    Label (178,803 103x24), "STEP 08"
    RoundedRectangle (285,800 125x30)
    RoundedRectangle (420,800 454x30)
    RoundedRectangle (157,856 762x64)
    Label (178,876 103x24), "STEP 09"
    RoundedRectangle (285,873 125x30)
    RoundedRectangle (420,873 454x30)
    RoundedRectangle (157,929 762x64)
    Label (178,949 103x24), "STEP 10"
    RoundedRectangle (285,946 125x30)
    RoundedRectangle (420,946 454x30)
    RoundedRectangle (1000,272 762x64)
    Label (1021,292 103x24), "STEP 11"
    RoundedRectangle (1128,289 125x30)
    RoundedRectangle (1263,289 454x30)
    RoundedRectangle (1000,345 762x64)
    Label (1021,365 103x24), "STEP 12"
    RoundedRectangle (1128,362 125x30)
    RoundedRectangle (1263,362 454x30)
    RoundedRectangle (1000,418 762x64)
    Label (1021,438 103x24), "STEP 13"
    RoundedRectangle (1128,435 125x30)
    RoundedRectangle (1263,435 454x30)
    RoundedRectangle (1000,491 762x64)
    Label (1021,511 103x24), "STEP 14"
    RoundedRectangle (1128,508 125x30)
    RoundedRectangle (1263,508 454x30)
    RoundedRectangle (1000,564 762x64)
    Label (1021,584 103x24), "STEP 15"
    RoundedRectangle (1128,581 125x30)
    RoundedRectangle (1263,581 454x30)
    RoundedRectangle (1000,637 762x64)
    Label (1021,657 103x24), "STEP 16"
    RoundedRectangle (1128,654 125x30)
    RoundedRectangle (1263,654 454x30)
    RoundedRectangle (1000,710 762x64)
    Label (1021,730 103x24), "STEP 17"
    RoundedRectangle (1128,727 125x30)
    RoundedRectangle (1263,727 454x30)
    RoundedRectangle (1000,783 762x64)
    Label (1021,803 103x24), "STEP 18"
    RoundedRectangle (1128,800 125x30)
    RoundedRectangle (1263,800 454x30)
    RoundedRectangle (1000,856 762x64)
    Label (1021,876 103x24), "STEP 19"
    RoundedRectangle (1128,873 125x30)
    RoundedRectangle (1263,873 454x30)
    RoundedRectangle (1000,929 762x64)
    Label (1021,949 103x24), "STEP 20"
    RoundedRectangle (1128,946 125x30)
    RoundedRectangle (1263,946 454x30)
    Rectangle (758,175 403x30), "RECIPE OVERVIEW"
    RoundedRectangle (703,219 587x34)
    RoundedRectangle (833,221 454x30)
    ComboBoxInteger (713,221 112x30)
    Label (628,224 103x24), "RECIPE"
    Group (1828,25 45x45)
        OnMouseClick: toggle HMI_Ctrl.MenuButton
        RoundedRectangle (0,0 45x45), colour toggle: HMI_Ctrl.MenuButton
        Image (6,5 33x35), image: ImagePool.Menu Button
    Group (1604,113 269x41)
        RoundedRectangle (0,1 269x39)
        Label (1,0 108x41), "OVERVIEW"
        Label (161,0 105x41), "EDIT RECIPE"
        Group (111,6 47x26)
            OnMouseClick: change screen: RecipeSSUR_Page
            Group (0,0 47x26)
                Ellipse (0,0 26x26)
                Ellipse (21,0 26x26)
                RoundedRectangle (8,0 29x26)
            Ellipse (1,1 24x24)
            Ellipse (23,1 23x24)
            RoundedRectangle (9,1 28x24)
            Ellipse (5,5 17x17)
    Frame (0,840 1918x221), invisible if: HMI_Ctrl.CloseMenuButton
        shows Popup_MenuPage()
END_VISUALIZATION

